RoboDK station: Config_1NewDrillbit.rdk

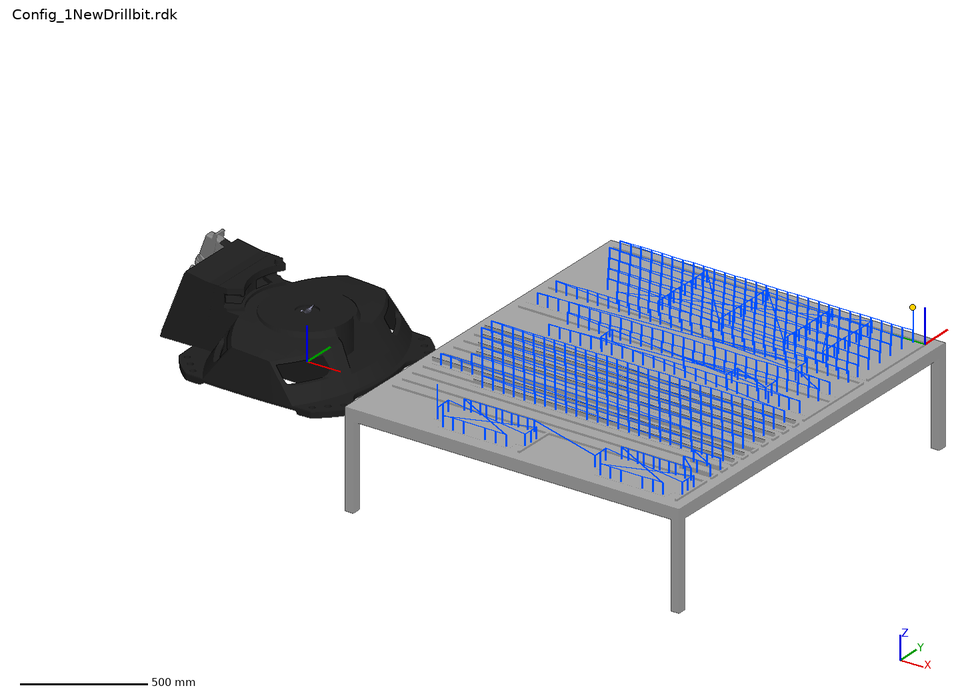
[picture v0: the station drawn from its stored meshes, robots at their saved joint values, targets as dots, program paths as lines]
Station Config_1NewDrillbit (saved by RoboDK 5.2.3). Poses are relative to the parent item; angles as X-Y-Z fixed-axis rotations.
  - frame KUKA KR 210 R2700 extra Base at (0, 0, 0) mm
    - robot KUKA KR 210 R2700 extra: 6 axes, payload 210 kg, reach 2696 mm, repeatability 0.06 mm, weight 1068 kg
        joint limits [-185, -140, -120, -350, -125, -350] to [185, -5, 155, 350, 125, 350]; home [0, -90, 90, 0, 0, 0]; saved at [43.451, -82.307, 119.902, -52.09, 33.269, 83.395]
      - tool Spindle, TCP at (32, 0, 260) mm, rotated rx 0 ry 39 rz 0 deg, size 157.3 x 72 x 259.9 mm
  - frame Corner First Plate at (2495, 660, 510.8) mm, rotated rx 0 ry 0 rz 90 deg
  - object Table 1 at (1700, -800, 455) mm, rotated rx 0 ry 0 rz 90 deg, size 1820 x 1600 x 475 mm, geometry from Table 1.stl
  - machining project Path1 settings: rotZ(0) | rotX(0)*rotY(0) | rotz(0) | onStart | onPathStart | onApproach | onPoint | onRetract | onFinish | SetRPM(%1) | SetTool(%1) | Extruder(%1) | default | default | OutOnMov(%1) | OutOffMov(%1) | onPathFinish | M_RunCode(%1)
  - program Path1 (1722 instructions, listed below)
  - object Config_1 at (2495, 660, 510.8) mm, rotated rx 0 ry 0 rz 90 deg
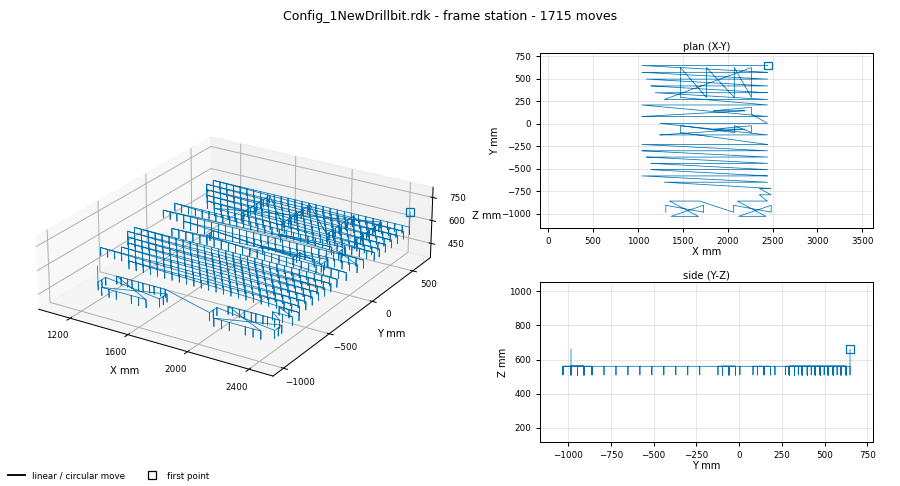
[picture p0: tool path of Config_1NewDrillbit.rdk in frame station, 1715 of 1715 moves have a stored position in this frame; points joined in program order, loops and branches not executed]

--- program Path1 (robot KUKA KR 210 R2700 extra) ---
  Smooth(1)
  Set speed (1000.0 mm/s)
  Set Ref.: Corner First Plate
  Set Tool: Spindle
  Show Spindle
  MoveJ 1 to (-10.8, 50, 150) mm, rotated rx -180 ry 0 rz 90 deg; joints [-16.649, -45.763, 65.757, 18.983, 33.662, -29.06]
  MoveL 2 to (-10.8, 50, 150) mm, rotated rx -180 ry 0 rz 90 deg; joints [-16.649, -45.763, 65.757, 18.983, 33.662, -29.06]
  MoveL 3 to (-10.8, 50, 50) mm, rotated rx -180 ry 0 rz 90 deg; joints [-16.649, -43.604, 67.207, 20.959, 30.27, -31.388]
  MoveL 4 to (-10.8, 50, 50) mm, rotated rx -180 ry 0 rz 90 deg; joints [-16.649, -43.604, 67.207, 20.959, 30.27, -31.388]
  Set speed (150.0 mm/s)
  MoveL 5 to (-10.8, 50, -0.5) mm, rotated rx 180 ry 0 rz 90 deg; joints [-16.649, -42.408, 67.766, 22.1, 28.636, -32.698]
  MoveL 6 to (-10.8, 50, 50) mm, rotated rx -180 ry 0 rz 90 deg; joints [-16.649, -43.604, 67.207, 20.959, 30.27, -31.388]
  MoveL 7 to (-10.8, 100, 50) mm, rotated rx 180 ry 0 rz 90 deg; joints [-17.019, -45.861, 71.178, 22.478, 28.801, -33.31]
  MoveL 8 to (-10.8, 100, -0.5) mm, rotated rx -180 ry 0 rz 90 deg; joints [-17.019, -44.622, 71.724, 23.798, 27.159, -34.805]
  MoveL 9 to (-10.8, 100, 50) mm, rotated rx 180 ry 0 rz 90 deg; joints [-17.019, -45.861, 71.178, 22.478, 28.801, -33.31]
  MoveL 10 to (-10.8, 150, 50) mm, rotated rx 180 ry 0 rz 90 deg; joints [-17.405, -48.034, 74.962, 24.095, 27.459, -35.336]
  MoveL 11 to (-10.8, 150, -0.5) mm, rotated rx 180 ry 0 rz 90 deg; joints [-17.405, -46.752, 75.499, 25.62, 25.808, -37.042]
  MoveL 12 to (-10.8, 150, 50) mm, rotated rx 180 ry 0 rz 90 deg; joints [-17.405, -48.034, 74.962, 24.095, 27.459, -35.336]
  MoveL 13 to (-10.8, 200, 50) mm, rotated rx -180 ry 0 rz 90 deg; joints [-17.809, -50.139, 78.585, 25.814, 26.233, -37.473]
  MoveL 14 to (-10.8, 200, -0.5) mm, rotated rx -180 ry 0 rz 90 deg; joints [-17.809, -48.813, 79.116, 27.569, 24.574, -39.416]
  MoveL 15 to (-10.8, 200, 50) mm, rotated rx -180 ry 0 rz 90 deg; joints [-17.809, -50.139, 78.585, 25.814, 26.233, -37.473]
  MoveL 16 to (-10.8, 250, 50) mm, rotated rx 180 ry 0 rz 90 deg; joints [-18.231, -52.185, 82.068, 27.636, 25.116, -39.724]
  MoveL 17 to (-10.8, 250, -0.5) mm, rotated rx 180 ry 0 rz 90 deg; joints [-18.231, -50.816, 82.594, 29.651, 23.452, -41.933]
  MoveL 18 to (-10.8, 250, 50) mm, rotated rx 180 ry 0 rz 90 deg; joints [-18.231, -52.185, 82.068, 27.636, 25.116, -39.724]
  MoveL 19 to (-10.8, 300, 50) mm, rotated rx -180 ry 0 rz 90 deg; joints [-18.673, -54.184, 85.426, 29.563, 24.104, -42.09]
  MoveL 20 to (-10.8, 300, -0.5) mm, rotated rx -180 ry 0 rz 90 deg; joints [-18.673, -52.769, 85.95, 31.865, 22.437, -44.595]
  MoveL 21 to (-10.8, 300, 50) mm, rotated rx -180 ry 0 rz 90 deg; joints [-18.673, -54.184, 85.426, 29.563, 24.104, -42.09]
  MoveL 22 to (-10.8, 350, 50) mm, rotated rx 180 ry 0 rz 90 deg; joints [-19.136, -56.141, 88.674, 31.59, 23.193, -44.569]
  MoveL 23 to (-10.8, 350, -0.5) mm, rotated rx 180 ry 0 rz 90 deg; joints [-19.136, -54.681, 89.197, 34.21, 21.527, -47.403]
  MoveL 24 to (-10.8, 350, 50) mm, rotated rx 180 ry 0 rz 90 deg; joints [-19.136, -56.141, 88.674, 31.59, 23.193, -44.569]
  MoveL 25 to (-10.8, 400, 50) mm, rotated rx -180 ry 0 rz 90 deg; joints [-19.622, -58.066, 91.821, 33.711, 22.382, -47.158]
  MoveL 26 to (-10.8, 400, -0.5) mm, rotated rx 180 ry 0 rz 90 deg; joints [-19.622, -56.557, 92.346, 36.679, 20.72, -50.348]
  MoveL 27 to (-10.8, 400, 50) mm, rotated rx -180 ry 0 rz 90 deg; joints [-19.622, -58.066, 91.821, 33.711, 22.382, -47.158]
  MoveL 28 to (-10.8, 450, 50) mm, rotated rx 180 ry 0 rz 90 deg; joints [-20.132, -59.962, 94.878, 35.915, 21.67, -49.846]
  MoveL 29 to (-10.8, 450, -0.5) mm, rotated rx -180 ry 0 rz 90 deg; joints [-20.132, -58.404, 95.405, 39.258, 20.016, -53.422]
  MoveL 30 to (-10.8, 450, 50) mm, rotated rx 180 ry 0 rz 90 deg; joints [-20.132, -59.962, 94.878, 35.915, 21.67, -49.846]
  MoveL 31 to (-10.8, 500, 50) mm, rotated rx 180 ry 0 rz 90 deg; joints [-20.668, -61.836, 97.851, 38.189, 21.056, -52.621]
  MoveL 32 to (-10.8, 500, -0.5) mm, rotated rx -180 ry 0 rz 90 deg; joints [-20.668, -60.227, 98.383, 41.928, 19.416, -56.606]
  MoveL 33 to (-10.8, 500, 50) mm, rotated rx 180 ry 0 rz 90 deg; joints [-20.668, -61.836, 97.851, 38.189, 21.056, -52.621]
  MoveL 34 to (-10.8, 550, 50) mm, rotated rx -180 ry 0 rz 90 deg; joints [-21.232, -63.693, 100.748, 40.512, 20.539, -55.465]
  MoveL 35 to (-10.8, 550, -0.5) mm, rotated rx 180 ry 0 rz 90 deg; joints [-21.232, -62.029, 101.285, 44.666, 18.917, -59.878]
  MoveL 36 to (-10.8, 550, 50) mm, rotated rx -180 ry 0 rz 90 deg; joints [-21.232, -63.693, 100.748, 40.512, 20.539, -55.465]
  MoveL 37 to (-10.8, 600, 50) mm, rotated rx 180 ry 0 rz 90 deg; joints [-21.826, -65.537, 103.573, 42.861, 20.119, -58.356]
  MoveL 38 to (-10.8, 600, -0.5) mm, rotated rx 180 ry 0 rz 90 deg; joints [-21.826, -63.817, 104.117, 47.441, 18.521, -63.209]
  MoveL 39 to (-10.8, 600, 50) mm, rotated rx 180 ry 0 rz 90 deg; joints [-21.826, -65.537, 103.573, 42.861, 20.119, -58.356]
  MoveL 40 to (-10.8, 650, 50) mm, rotated rx -180 ry 0 rz 90 deg; joints [-22.453, -67.372, 106.331, 45.208, 19.797, -61.269]
  MoveL 41 to (-10.8, 650, -0.5) mm, rotated rx 180 ry 0 rz 90 deg; joints [-22.453, -65.593, 106.883, 50.215, 18.227, -66.564]
  MoveL 42 to (-10.8, 650, 50) mm, rotated rx -180 ry 0 rz 90 deg; joints [-22.453, -67.372, 106.331, 45.208, 19.797, -61.269]
  MoveL 43 to (-10.8, 700, 50) mm, rotated rx -180 ry 0 rz 90 deg; joints [-23.115, -69.203, 109.025, 47.523, 19.571, -64.173]
  MoveL 44 to (-10.8, 700, -0.5) mm, rotated rx 180 ry 0 rz 90 deg; joints [-23.115, -67.362, 109.587, 52.95, 18.032, -69.905]
  MoveL 45 to (-10.8, 700, 50) mm, rotated rx -180 ry 0 rz 90 deg; joints [-23.115, -69.203, 109.025, 47.523, 19.571, -64.173]
  MoveL 46 to (-10.8, 750, 50) mm, rotated rx -180 ry 0 rz 90 deg; joints [-23.814, -71.033, 111.66, 49.773, 19.44, -67.039]
  MoveL 47 to (-10.8, 750, -0.5) mm, rotated rx 180 ry 0 rz 90 deg; joints [-23.814, -69.127, 112.233, 55.604, 17.936, -73.194]
  MoveL 48 to (-10.8, 750, 50) mm, rotated rx -180 ry 0 rz 90 deg; joints [-23.814, -71.033, 111.66, 49.773, 19.44, -67.039]
  MoveL 49 to (-10.8, 800, 50) mm, rotated rx -180 ry 0 rz 90 deg; joints [-24.555, -72.867, 114.238, 51.923, 19.404, -69.834]
  MoveL 50 to (-10.8, 800, -0.5) mm, rotated rx -180 ry 0 rz 90 deg; joints [-24.555, -70.893, 114.823, 58.134, 17.935, -76.388]
  MoveL 51 to (-10.8, 800, 50) mm, rotated rx -180 ry 0 rz 90 deg; joints [-24.555, -72.867, 114.238, 51.923, 19.404, -69.834]
  MoveL 52 to (-10.8, 850, 50) mm, rotated rx 180 ry 0 rz 90 deg; joints [-25.34, -74.708, 116.76, 53.942, 19.461, -72.529]
  MoveL 53 to (-10.8, 850, -0.5) mm, rotated rx 180 ry 0 rz 90 deg; joints [-25.34, -72.662, 117.358, 60.5, 18.027, -79.453]
  MoveL 54 to (-10.8, 850, 50) mm, rotated rx 180 ry 0 rz 90 deg; joints [-25.34, -74.708, 116.76, 53.942, 19.461, -72.529]
  MoveL 55 to (-10.8, 900, 50) mm, rotated rx -180 ry 0 rz 90 deg; joints [-26.173, -76.561, 119.228, 55.798, 19.61, -75.093]
  MoveL 56 to (-10.8, 900, -0.5) mm, rotated rx -180 ry 0 rz 90 deg; joints [-26.173, -74.439, 119.842, 62.666, 18.208, -82.352]
  MoveL 57 to (-10.8, 900, 50) mm, rotated rx -180 ry 0 rz 90 deg; joints [-26.173, -76.561, 119.228, 55.798, 19.61, -75.093]
  MoveL 58 to (-10.8, 950, 50) mm, rotated rx -180 ry 0 rz 90 deg; joints [-27.058, -78.43, 121.643, 57.462, 19.851, -77.502]
  MoveL 59 to (-10.8, 950, -0.5) mm, rotated rx 180 ry 0 rz 90 deg; joints [-27.058, -76.227, 122.274, 64.602, 18.476, -85.059]
  MoveL 60 to (-10.8, 950, 50) mm, rotated rx -180 ry 0 rz 90 deg; joints [-27.058, -78.43, 121.643, 57.462, 19.851, -77.502]
  MoveL 61 to (-10.8, 1000, 50) mm, rotated rx 180 ry 0 rz 90 deg; joints [-28.001, -80.318, 124.007, 58.912, 20.182, -79.735]
  MoveL 62 to (-10.8, 1000, -0.5) mm, rotated rx 180 ry 0 rz 90 deg; joints [-28.001, -78.031, 124.656, 66.28, 18.827, -87.549]
  MoveL 63 to (-10.8, 1000, 50) mm, rotated rx 180 ry 0 rz 90 deg; joints [-28.001, -80.318, 124.007, 58.912, 20.182, -79.735]
  MoveL 64 to (-10.8, 1050, 50) mm, rotated rx -180 ry 0 rz 90 deg; joints [-29.005, -82.231, 126.318, 60.129, 20.604, -81.776]
  MoveL 65 to (-10.8, 1050, -0.5) mm, rotated rx 180 ry 0 rz 90 deg; joints [-29.005, -79.854, 126.988, 67.681, 19.26, -89.808]
  MoveL 66 to (-10.8, 1050, 50) mm, rotated rx -180 ry 0 rz 90 deg; joints [-29.005, -82.231, 126.318, 60.129, 20.604, -81.776]
  MoveL 67 to (-10.8, 1100, 50) mm, rotated rx 180 ry 0 rz 90 deg; joints [-30.078, -84.172, 128.578, 61.097, 21.117, -83.613]
  MoveL 68 to (-10.8, 1100, -0.5) mm, rotated rx 180 ry 0 rz 90 deg; joints [-30.078, -81.701, 129.27, 68.792, 19.774, -91.823]
  MoveL 69 to (-10.8, 1100, 50) mm, rotated rx 180 ry 0 rz 90 deg; joints [-30.078, -84.172, 128.578, 61.097, 21.117, -83.613]
  MoveL 70 to (-10.8, 1150, 50) mm, rotated rx -180 ry 0 rz 90 deg; joints [-31.224, -86.147, 130.785, 61.808, 21.724, -85.24]
  MoveL 71 to (-10.8, 1150, -0.5) mm, rotated rx 180 ry 0 rz 90 deg; joints [-31.224, -83.576, 131.502, 69.603, 20.368, -93.59]
  MoveL 72 to (-10.8, 1150, 50) mm, rotated rx -180 ry 0 rz 90 deg; joints [-31.224, -86.147, 130.785, 61.808, 21.724, -85.24]
  MoveL 73 to (-10.8, 1200, 50) mm, rotated rx 180 ry 0 rz 90 deg; joints [-32.452, -88.16, 132.937, 62.257, 22.43, -86.657]
  MoveL 74 to (-10.8, 1200, -0.5) mm, rotated rx 180 ry 0 rz 90 deg; joints [-32.452, -85.485, 133.681, 70.11, 21.045, -95.109]
  MoveL 75 to (-10.8, 1200, 50) mm, rotated rx 180 ry 0 rz 90 deg; joints [-32.452, -88.16, 132.937, 62.257, 22.43, -86.657]
  MoveL 76 to (-10.8, 1250, 50) mm, rotated rx 180 ry 0 rz 90 deg; joints [-33.768, -90.216, 135.034, 62.444, 23.238, -87.866]
  MoveL 77 to (-10.8, 1250, -0.5) mm, rotated rx 180 ry 0 rz 90 deg; joints [-33.768, -87.431, 135.807, 70.315, 21.808, -96.384]
  MoveL 78 to (-10.8, 1250, 50) mm, rotated rx 180 ry 0 rz 90 deg; joints [-33.768, -90.216, 135.034, 62.444, 23.238, -87.866]
  MoveL 79 to (-10.8, 1300, 50) mm, rotated rx 180 ry 0 rz 90 deg; joints [-35.181, -92.32, 137.073, 62.376, 24.157, -88.879]
  MoveL 80 to (-10.8, 1300, -0.5) mm, rotated rx -180 ry 0 rz 90 deg; joints [-35.181, -89.419, 137.878, 70.222, 22.664, -97.425]
  MoveL 81 to (-10.8, 1300, 50) mm, rotated rx 180 ry 0 rz 90 deg; joints [-35.181, -92.32, 137.073, 62.376, 24.157, -88.879]
  MoveL 82 to (-10.8, 1350, 50) mm, rotated rx -180 ry 0 rz 90 deg; joints [-36.701, -94.476, 139.051, 62.061, 25.197, -89.708]
  MoveL 83 to (-10.8, 1350, -0.5) mm, rotated rx -180 ry 0 rz 90 deg; joints [-36.701, -91.455, 139.89, 69.839, 23.619, -98.245]
  MoveL 84 to (-10.8, 1350, 50) mm, rotated rx -180 ry 0 rz 90 deg; joints [-36.701, -94.476, 139.051, 62.061, 25.197, -89.708]
  MoveL 85 to (-10.8, 1400, 50) mm, rotated rx -180 ry 0 rz 90 deg; joints [-38.337, -96.689, 140.964, 61.514, 26.367, -90.372]
  MoveL 86 to (-10.8, 1400, -0.5) mm, rotated rx 180 ry 0 rz 90 deg; joints [-38.337, -93.543, 141.842, 69.179, 24.685, -98.863]
  MoveL 87 to (-10.8, 1400, 50) mm, rotated rx -180 ry 0 rz 90 deg; joints [-38.337, -96.689, 140.964, 61.514, 26.367, -90.372]
  MoveL 88 to (-10.8, 1450, 50) mm, rotated rx -180 ry 0 rz 90 deg; joints [-40.1, -98.961, 142.81, 60.755, 27.683, -90.897]
  MoveL 89 to (-10.8, 1450, -0.5) mm, rotated rx -180 ry 0 rz 90 deg; joints [-40.1, -95.687, 143.728, 68.26, 25.874, -99.3]
  MoveL 90 to (-10.8, 1450, 50) mm, rotated rx -180 ry 0 rz 90 deg; joints [-40.1, -98.961, 142.81, 60.755, 27.683, -90.897]
  MoveL 91 to (-86.48, 50, 50) mm, rotated rx 180 ry 0 rz 90 deg; joints [-14.798, -44.582, 68.933, 19.373, 28.984, -28.699]
  MoveL 92 to (-86.48, 50, -0.5) mm, rotated rx 180 ry 0 rz 90 deg; joints [-14.798, -43.367, 69.486, 20.5, 27.322, -29.977]
  MoveL 93 to (-86.48, 50, 50) mm, rotated rx 180 ry 0 rz 90 deg; joints [-14.798, -44.582, 68.933, 19.373, 28.984, -28.699]
  MoveL 94 to (-86.48, 100, 50) mm, rotated rx 180 ry 0 rz 90 deg; joints [-15.131, -46.823, 72.859, 20.836, 27.506, -30.521]
  MoveL 95 to (-86.48, 100, -0.5) mm, rotated rx -180 ry 0 rz 90 deg; joints [-15.131, -45.565, 73.401, 22.149, 25.831, -31.99]
  MoveL 96 to (-86.48, 100, 50) mm, rotated rx 180 ry 0 rz 90 deg; joints [-15.131, -46.823, 72.859, 20.836, 27.506, -30.521]
  MoveL 97 to (-86.48, 150, 50) mm, rotated rx -180 ry 0 rz 90 deg; joints [-15.479, -48.988, 76.608, 22.405, 26.146, -32.455]
  MoveL 98 to (-86.48, 150, -0.5) mm, rotated rx -180 ry 0 rz 90 deg; joints [-15.479, -47.686, 77.142, 23.933, 24.459, -34.144]
  MoveL 99 to (-86.48, 150, 50) mm, rotated rx -180 ry 0 rz 90 deg; joints [-15.479, -48.988, 76.608, 22.405, 26.146, -32.455]
  MoveL 100 to (-86.48, 200, 50) mm, rotated rx -180 ry 0 rz 90 deg; joints [-15.843, -51.088, 80.205, 24.086, 24.897, -34.509]
  MoveL 101 to (-86.48, 200, -0.5) mm, rotated rx 180 ry 0 rz 90 deg; joints [-15.843, -49.742, 80.734, 25.859, 23.198, -36.45]
  MoveL 102 to (-86.48, 200, 50) mm, rotated rx -180 ry 0 rz 90 deg; joints [-15.843, -51.088, 80.205, 24.086, 24.897, -34.509]
  MoveL 103 to (-86.48, 250, 50) mm, rotated rx 180 ry 0 rz 90 deg; joints [-16.224, -53.135, 83.669, 25.883, 23.753, -36.689]
  MoveL 104 to (-86.48, 250, -0.5) mm, rotated rx -180 ry 0 rz 90 deg; joints [-16.224, -51.744, 84.194, 27.935, 22.045, -38.917]
  MoveL 105 to (-86.48, 250, 50) mm, rotated rx 180 ry 0 rz 90 deg; joints [-16.224, -53.135, 83.669, 25.883, 23.753, -36.689]
  MoveL 106 to (-86.48, 300, 50) mm, rotated rx -180 ry 0 rz 90 deg; joints [-16.624, -55.137, 87.014, 27.798, 22.709, -38.998]
  MoveL 107 to (-86.48, 300, -0.5) mm, rotated rx 180 ry 0 rz 90 deg; joints [-16.624, -53.701, 87.537, 30.167, 20.994, -41.55]
  MoveL 108 to (-86.48, 300, 50) mm, rotated rx -180 ry 0 rz 90 deg; joints [-16.624, -55.137, 87.014, 27.798, 22.709, -38.998]
  MoveL 109 to (-86.48, 350, 50) mm, rotated rx 180 ry 0 rz 90 deg; joints [-17.042, -57.103, 90.253, 29.831, 21.764, -41.437]
  MoveL 110 to (-86.48, 350, -0.5) mm, rotated rx 180 ry 0 rz 90 deg; joints [-17.042, -55.619, 90.777, 32.555, 20.045, -44.353]
  MoveL 111 to (-86.48, 350, 50) mm, rotated rx 180 ry 0 rz 90 deg; joints [-17.042, -57.103, 90.253, 29.831, 21.764, -41.437]
  MoveL 112 to (-86.48, 400, 50) mm, rotated rx 180 ry 0 rz 90 deg; joints [-17.482, -59.039, 93.396, 31.978, 20.915, -44.004]
  MoveL 113 to (-86.48, 400, -0.5) mm, rotated rx 180 ry 0 rz 90 deg; joints [-17.482, -57.506, 93.922, 35.095, 19.197, -47.323]
  MoveL 114 to (-86.48, 400, 50) mm, rotated rx 180 ry 0 rz 90 deg; joints [-17.482, -59.039, 93.396, 31.978, 20.915, -44.004]
  MoveL 115 to (-86.48, 450, 50) mm, rotated rx -180 ry 0 rz 90 deg; joints [-17.945, -60.951, 96.453, 34.23, 20.163, -46.692]
  MoveL 116 to (-86.48, 450, -0.5) mm, rotated rx 180 ry 0 rz 90 deg; joints [-17.945, -59.366, 96.983, 37.779, 18.451, -50.452]
  MoveL 117 to (-86.48, 450, 50) mm, rotated rx -180 ry 0 rz 90 deg; joints [-17.945, -60.951, 96.453, 34.23, 20.163, -46.692]
  MoveL 118 to (-86.48, 500, 50) mm, rotated rx 180 ry 0 rz 90 deg; joints [-18.431, -62.844, 99.43, 36.574, 19.507, -49.488]
  MoveL 119 to (-86.48, 500, -0.5) mm, rotated rx 180 ry 0 rz 90 deg; joints [-18.431, -61.206, 99.965, 40.589, 17.807, -53.725]
  MoveL 120 to (-86.48, 500, 50) mm, rotated rx 180 ry 0 rz 90 deg; joints [-18.431, -62.844, 99.43, 36.574, 19.507, -49.488]
  MoveL 121 to (-86.48, 550, 50) mm, rotated rx 180 ry 0 rz 90 deg; joints [-18.944, -64.724, 102.334, 38.99, 18.948, -52.374]
  MoveL 122 to (-86.48, 550, -0.5) mm, rotated rx -180 ry 0 rz 90 deg; joints [-18.944, -63.029, 102.875, 43.499, 17.266, -57.118]
  MoveL 123 to (-86.48, 550, 50) mm, rotated rx 180 ry 0 rz 90 deg; joints [-18.944, -64.724, 102.334, 38.99, 18.948, -52.374]
  MoveL 124 to (-86.48, 600, 50) mm, rotated rx -180 ry 0 rz 90 deg; joints [-19.485, -66.595, 105.169, 41.455, 18.486, -55.329]
  MoveL 125 to (-86.48, 600, -0.5) mm, rotated rx -180 ry 0 rz 90 deg; joints [-19.485, -64.841, 105.718, 46.478, 16.828, -60.599]
  MoveL 126 to (-86.48, 600, 50) mm, rotated rx -180 ry 0 rz 90 deg; joints [-19.485, -66.595, 105.169, 41.455, 18.486, -55.329]
  MoveL 127 to (-86.48, 650, 50) mm, rotated rx 180 ry 0 rz 90 deg; joints [-20.056, -68.461, 107.941, 43.937, 18.122, -58.322]
  MoveL 128 to (-86.48, 650, -0.5) mm, rotated rx 180 ry 0 rz 90 deg; joints [-20.056, -66.646, 108.498, 49.483, 16.493, -64.13]
  MoveL 129 to (-86.48, 650, 50) mm, rotated rx 180 ry 0 rz 90 deg; joints [-20.056, -68.461, 107.941, 43.937, 18.122, -58.322]
  MoveL 130 to (-86.48, 700, 50) mm, rotated rx -180 ry 0 rz 90 deg; joints [-20.661, -70.327, 110.652, 46.401, 17.855, -61.321]
  MoveL 131 to (-86.48, 700, -0.5) mm, rotated rx 180 ry 0 rz 90 deg; joints [-20.661, -68.447, 111.22, 52.467, 16.26, -67.665]
  MoveL 132 to (-86.48, 700, 50) mm, rotated rx -180 ry 0 rz 90 deg; joints [-20.661, -70.327, 110.652, 46.401, 17.855, -61.321]
  MoveL 133 to (-86.48, 750, 50) mm, rotated rx -180 ry 0 rz 90 deg; joints [-21.301, -72.199, 113.306, 48.809, 17.686, -64.288]
  MoveL 134 to (-86.48, 750, -0.5) mm, rotated rx 180 ry 0 rz 90 deg; joints [-21.301, -70.25, 113.886, 55.379, 16.129, -71.153]
  MoveL 135 to (-86.48, 750, 50) mm, rotated rx -180 ry 0 rz 90 deg; joints [-21.301, -72.199, 113.306, 48.809, 17.686, -64.288]
  MoveL 136 to (-86.48, 800, 50) mm, rotated rx -180 ry 0 rz 90 deg; joints [-21.98, -74.079, 115.905, 51.119, 17.613, -67.184]
  MoveL 137 to (-86.48, 800, -0.5) mm, rotated rx -180 ry 0 rz 90 deg; joints [-21.98, -72.058, 116.499, 58.165, 16.096, -74.544]
  MoveL 138 to (-86.48, 800, 50) mm, rotated rx -180 ry 0 rz 90 deg; joints [-21.98, -74.079, 115.905, 51.119, 17.613, -67.184]
  MoveL 139 to (-86.48, 850, 50) mm, rotated rx 180 ry 0 rz 90 deg; joints [-22.702, -75.973, 118.452, 53.291, 17.635, -69.971]
  MoveL 140 to (-86.48, 850, -0.5) mm, rotated rx -180 ry 0 rz 90 deg; joints [-22.702, -73.875, 119.061, 60.773, 16.159, -77.789]
  MoveL 141 to (-86.48, 850, 50) mm, rotated rx 180 ry 0 rz 90 deg; joints [-22.702, -75.973, 118.452, 53.291, 17.635, -69.971]
  MoveL 142 to (-86.48, 900, 50) mm, rotated rx 180 ry 0 rz 90 deg; joints [-23.469, -77.886, 120.948, 55.285, 17.752, -72.611]
  MoveL 143 to (-86.48, 900, -0.5) mm, rotated rx 180 ry 0 rz 90 deg; joints [-23.469, -75.707, 121.574, 63.158, 16.314, -80.843]
  MoveL 144 to (-86.48, 900, 50) mm, rotated rx 180 ry 0 rz 90 deg; joints [-23.469, -77.886, 120.948, 55.285, 17.752, -72.611]
  MoveL 145 to (-86.48, 950, 50) mm, rotated rx -180 ry 0 rz 90 deg; joints [-24.288, -79.823, 123.395, 57.066, 17.964, -75.072]
  MoveL 146 to (-86.48, 950, -0.5) mm, rotated rx -180 ry 0 rz 90 deg; joints [-24.288, -77.558, 124.039, 65.278, 16.557, -83.669]
  MoveL 147 to (-86.48, 950, 50) mm, rotated rx -180 ry 0 rz 90 deg; joints [-24.288, -79.823, 123.395, 57.066, 17.964, -75.072]
  MoveL 148 to (-86.48, 1000, 50) mm, rotated rx -180 ry 0 rz 90 deg; joints [-25.161, -81.788, 125.791, 58.604, 18.268, -77.326]
  MoveL 149 to (-86.48, 1000, -0.5) mm, rotated rx 180 ry 0 rz 90 deg; joints [-25.161, -79.433, 126.457, 67.099, 16.885, -86.235]
  MoveL 150 to (-86.48, 1000, 50) mm, rotated rx -180 ry 0 rz 90 deg; joints [-25.161, -81.788, 125.791, 58.604, 18.268, -77.326]
  MoveL 151 to (-86.48, 1050, 50) mm, rotated rx -180 ry 0 rz 90 deg; joints [-26.095, -83.789, 128.139, 59.872, 18.666, -79.349]
  MoveL 152 to (-86.48, 1050, -0.5) mm, rotated rx -180 ry 0 rz 90 deg; joints [-26.095, -81.337, 128.827, 68.595, 17.297, -88.518]
  MoveL 153 to (-86.48, 1050, 50) mm, rotated rx -180 ry 0 rz 90 deg; joints [-26.095, -83.789, 128.139, 59.872, 18.666, -79.349]
  MoveL 154 to (-86.48, 1100, 50) mm, rotated rx 180 ry 0 rz 90 deg; joints [-27.096, -85.831, 130.438, 60.853, 19.16, -81.127]
  MoveL 155 to (-86.48, 1100, -0.5) mm, rotated rx -180 ry 0 rz 90 deg; joints [-27.096, -83.277, 131.151, 69.748, 17.79, -90.503]
  MoveL 156 to (-86.48, 1100, 50) mm, rotated rx 180 ry 0 rz 90 deg; joints [-27.096, -85.831, 130.438, 60.853, 19.16, -81.127]
  MoveL 157 to (-86.48, 1150, 50) mm, rotated rx -180 ry 0 rz 90 deg; joints [-28.17, -87.921, 132.686, 61.533, 19.753, -82.65]
  MoveL 158 to (-86.48, 1150, -0.5) mm, rotated rx -180 ry 0 rz 90 deg; joints [-28.17, -85.258, 133.427, 70.547, 18.366, -92.183]
  MoveL 159 to (-86.48, 1150, 50) mm, rotated rx -180 ry 0 rz 90 deg; joints [-28.17, -87.921, 132.686, 61.533, 19.753, -82.65]
  MoveL 160 to (-86.48, 1200, 50) mm, rotated rx 180 ry 0 rz 90 deg; joints [-29.325, -90.065, 134.884, 61.907, 20.45, -83.915]
  MoveL 161 to (-86.48, 1200, -0.5) mm, rotated rx 180 ry 0 rz 90 deg; joints [-29.325, -87.288, 135.655, 70.984, 19.027, -93.555]
  MoveL 162 to (-86.48, 1200, 50) mm, rotated rx 180 ry 0 rz 90 deg; joints [-29.325, -90.065, 134.884, 61.907, 20.45, -83.915]
  MoveL 163 to (-86.48, 1250, 50) mm, rotated rx 180 ry 0 rz 90 deg; joints [-30.57, -92.272, 137.028, 61.975, 21.259, -84.926]
  MoveL 164 to (-86.48, 1250, -0.5) mm, rotated rx 180 ry 0 rz 90 deg; joints [-30.57, -89.374, 137.832, 71.061, 19.778, -94.623]
  MoveL 165 to (-86.48, 1250, 50) mm, rotated rx 180 ry 0 rz 90 deg; joints [-30.57, -92.272, 137.028, 61.975, 21.259, -84.926]
  MoveL 166 to (-86.48, 1300, 50) mm, rotated rx 180 ry 0 rz 90 deg; joints [-31.913, -94.55, 139.117, 61.744, 22.19, -85.693]
  MoveL 167 to (-86.48, 1300, -0.5) mm, rotated rx -180 ry 0 rz 90 deg; joints [-31.913, -91.525, 139.957, 70.782, 20.629, -95.397]
  MoveL 168 to (-86.48, 1300, 50) mm, rotated rx 180 ry 0 rz 90 deg; joints [-31.913, -94.55, 139.117, 61.744, 22.19, -85.693]
  MoveL 169 to (-86.48, 1350, 50) mm, rotated rx 180 ry 0 rz 90 deg; joints [-33.365, -96.907, 141.147, 61.226, 23.258, -86.233]
  MoveL 170 to (-86.48, 1350, -0.5) mm, rotated rx -180 ry 0 rz 90 deg; joints [-33.365, -93.749, 142.028, 70.158, 21.589, -95.891]
  MoveL 171 to (-86.48, 1350, 50) mm, rotated rx 180 ry 0 rz 90 deg; joints [-33.365, -96.907, 141.147, 61.226, 23.258, -86.233]
  MoveL 172 to (-86.48, 1400, 50) mm, rotated rx -180 ry 0 rz 90 deg; joints [-34.939, -99.35, 143.114, 60.44, 24.478, -86.569]
  MoveL 173 to (-86.48, 1400, -0.5) mm, rotated rx -180 ry 0 rz 90 deg; joints [-34.939, -96.055, 144.039, 69.205, 22.676, -96.127]
  MoveL 174 to (-86.48, 1400, 50) mm, rotated rx -180 ry 0 rz 90 deg; joints [-34.939, -99.35, 143.114, 60.44, 24.478, -86.569]
  MoveL 175 to (-86.48, 1450, 50) mm, rotated rx 180 ry 0 rz 90 deg; joints [-36.646, -101.889, 145.015, 59.412, 25.871, -86.731]
  MoveL 176 to (-86.48, 1450, -0.5) mm, rotated rx -180 ry 0 rz 90 deg; joints [-36.646, -98.452, 145.988, 67.945, 23.909, -96.132]
  MoveL 177 to (-86.48, 1450, 50) mm, rotated rx 180 ry 0 rz 90 deg; joints [-36.646, -101.889, 145.015, 59.412, 25.871, -86.731]
  MoveL 178 to (-162.16, 50, 50) mm, rotated rx 180 ry 0 rz 90 deg; joints [-12.916, -45.433, 70.428, 17.535, 27.831, -25.717]
  MoveL 179 to (-162.16, 50, -0.5) mm, rotated rx 180 ry 0 rz 90 deg; joints [-12.916, -44.202, 70.977, 18.62, 26.139, -26.934]
  MoveL 180 to (-162.16, 50, 50) mm, rotated rx 180 ry 0 rz 90 deg; joints [-12.916, -45.433, 70.428, 17.535, 27.831, -25.717]
  MoveL 181 to (-162.16, 100, 50) mm, rotated rx 180 ry 0 rz 90 deg; joints [-13.21, -47.663, 74.318, 18.914, 26.337, -27.409]
  MoveL 182 to (-162.16, 100, -0.5) mm, rotated rx 180 ry 0 rz 90 deg; joints [-13.21, -46.388, 74.857, 20.187, 24.628, -28.819]
  MoveL 183 to (-162.16, 100, 50) mm, rotated rx 180 ry 0 rz 90 deg; joints [-13.21, -47.663, 74.318, 18.914, 26.337, -27.409]
  MoveL 184 to (-162.16, 150, 50) mm, rotated rx 180 ry 0 rz 90 deg; joints [-13.517, -49.821, 78.04, 20.404, 24.955, -29.218]
  MoveL 185 to (-162.16, 150, -0.5) mm, rotated rx 180 ry 0 rz 90 deg; joints [-13.517, -48.502, 78.572, 21.897, 23.23, -30.854]
  MoveL 186 to (-162.16, 150, 50) mm, rotated rx 180 ry 0 rz 90 deg; joints [-13.517, -49.821, 78.04, 20.404, 24.955, -29.218]
  MoveL 187 to (-162.16, 200, 50) mm, rotated rx 180 ry 0 rz 90 deg; joints [-13.839, -51.919, 81.617, 22.012, 23.679, -31.154]
  MoveL 188 to (-162.16, 200, -0.5) mm, rotated rx 180 ry 0 rz 90 deg; joints [-13.839, -50.556, 82.144, 23.761, 21.937, -33.051]
  MoveL 189 to (-162.16, 200, 50) mm, rotated rx 180 ry 0 rz 90 deg; joints [-13.839, -51.919, 81.617, 22.012, 23.679, -31.154]
  MoveL 190 to (-162.16, 250, 50) mm, rotated rx 180 ry 0 rz 90 deg; joints [-14.176, -53.968, 85.066, 23.747, 22.502, -33.225]
  MoveL 191 to (-162.16, 250, -0.5) mm, rotated rx 180 ry 0 rz 90 deg; joints [-14.176, -52.558, 85.59, 25.791, 20.746, -35.423]
  MoveL 192 to (-162.16, 250, 50) mm, rotated rx 180 ry 0 rz 90 deg; joints [-14.176, -53.968, 85.066, 23.747, 22.502, -33.225]
  MoveL 193 to (-162.16, 300, 50) mm, rotated rx -180 ry 0 rz 90 deg; joints [-14.529, -55.976, 88.401, 25.613, 21.422, -35.437]
  MoveL 194 to (-162.16, 300, -0.5) mm, rotated rx 180 ry 0 rz 90 deg; joints [-14.529, -54.519, 88.924, 27.996, 19.654, -37.983]
  MoveL 195 to (-162.16, 300, 50) mm, rotated rx -180 ry 0 rz 90 deg; joints [-14.529, -55.976, 88.401, 25.613, 21.422, -35.437]
  MoveL 196 to (-162.16, 350, 50) mm, rotated rx 180 ry 0 rz 90 deg; joints [-14.901, -57.951, 91.634, 27.612, 20.435, -37.795]
  MoveL 197 to (-162.16, 350, -0.5) mm, rotated rx -180 ry 0 rz 90 deg; joints [-14.901, -56.445, 92.159, 30.385, 18.659, -40.737]
  MoveL 198 to (-162.16, 350, 50) mm, rotated rx 180 ry 0 rz 90 deg; joints [-14.901, -57.951, 91.634, 27.612, 20.435, -37.795]
  MoveL 199 to (-162.16, 400, 50) mm, rotated rx 180 ry 0 rz 90 deg; joints [-15.291, -59.898, 94.776, 29.745, 19.542, -40.299]
  MoveL 200 to (-162.16, 400, -0.5) mm, rotated rx 180 ry 0 rz 90 deg; joints [-15.291, -58.342, 95.304, 32.958, 17.762, -43.689]
  MoveL 201 to (-162.16, 400, 50) mm, rotated rx 180 ry 0 rz 90 deg; joints [-15.291, -59.898, 94.776, 29.745, 19.542, -40.299]
  MoveL 202 to (-162.16, 450, 50) mm, rotated rx -180 ry 0 rz 90 deg; joints [-15.702, -61.826, 97.835, 32.007, 18.743, -42.945]
  MoveL 203 to (-162.16, 450, -0.5) mm, rotated rx -180 ry 0 rz 90 deg; joints [-15.702, -60.216, 98.366, 35.712, 16.964, -46.837]
  MoveL 204 to (-162.16, 450, 50) mm, rotated rx -180 ry 0 rz 90 deg; joints [-15.702, -61.826, 97.835, 32.007, 18.743, -42.945]
  MoveL 205 to (-162.16, 500, 50) mm, rotated rx 180 ry 0 rz 90 deg; joints [-16.134, -63.737, 100.817, 34.388, 18.038, -45.725]
  MoveL 206 to (-162.16, 500, -0.5) mm, rotated rx 180 ry 0 rz 90 deg; joints [-16.134, -62.073, 101.354, 38.635, 16.266, -50.169]
  MoveL 207 to (-162.16, 500, 50) mm, rotated rx 180 ry 0 rz 90 deg; joints [-16.134, -63.737, 100.817, 34.388, 18.038, -45.725]
  MoveL 208 to (-162.16, 550, 50) mm, rotated rx 180 ry 0 rz 90 deg; joints [-16.591, -65.639, 103.728, 36.869, 17.427, -48.622]
  MoveL 209 to (-162.16, 550, -0.5) mm, rotated rx 180 ry 0 rz 90 deg; joints [-16.591, -63.916, 104.273, 41.703, 15.671, -53.664]
  MoveL 210 to (-162.16, 550, 50) mm, rotated rx 180 ry 0 rz 90 deg; joints [-16.591, -65.639, 103.728, 36.869, 17.427, -48.622]
  MoveL 211 to (-162.16, 600, 50) mm, rotated rx 180 ry 0 rz 90 deg; joints [-17.073, -67.536, 106.574, 39.426, 16.914, -51.614]
  MoveL 212 to (-162.16, 600, -0.5) mm, rotated rx -180 ry 0 rz 90 deg; joints [-17.073, -65.752, 107.127, 44.883, 15.179, -57.29]
  MoveL 213 to (-162.16, 600, 50) mm, rotated rx 180 ry 0 rz 90 deg; joints [-17.073, -67.536, 106.574, 39.426, 16.914, -51.614]
  MoveL 214 to (-162.16, 650, 50) mm, rotated rx 180 ry 0 rz 90 deg; joints [-17.584, -69.432, 109.359, 42.029, 16.497, -54.669]
  MoveL 215 to (-162.16, 650, -0.5) mm, rotated rx 180 ry 0 rz 90 deg; joints [-17.584, -67.583, 109.922, 48.13, 14.792, -61.005]
  MoveL 216 to (-162.16, 650, 50) mm, rotated rx 180 ry 0 rz 90 deg; joints [-17.584, -69.432, 109.359, 42.029, 16.497, -54.669]
  MoveL 217 to (-162.16, 700, 50) mm, rotated rx 180 ry 0 rz 90 deg; joints [-18.124, -71.333, 112.086, 44.636, 16.179, -57.751]
  MoveL 218 to (-162.16, 700, -0.5) mm, rotated rx -180 ry 0 rz 90 deg; joints [-18.124, -69.416, 112.661, 51.39, 14.509, -64.753]
  MoveL 219 to (-162.16, 700, 50) mm, rotated rx 180 ry 0 rz 90 deg; joints [-18.124, -71.333, 112.086, 44.636, 16.179, -57.751]
  MoveL 220 to (-162.16, 750, 50) mm, rotated rx 180 ry 0 rz 90 deg; joints [-18.698, -73.244, 114.759, 47.204, 15.959, -60.817]
  MoveL 221 to (-162.16, 750, -0.5) mm, rotated rx -180 ry 0 rz 90 deg; joints [-18.698, -71.255, 115.347, 54.597, 14.331, -68.474]
  MoveL 222 to (-162.16, 750, 50) mm, rotated rx 180 ry 0 rz 90 deg; joints [-18.698, -73.244, 114.759, 47.204, 15.959, -60.817]
  MoveL 223 to (-162.16, 800, 50) mm, rotated rx 180 ry 0 rz 90 deg; joints [-19.308, -75.169, 117.38, 49.683, 15.837, -63.817]
  MoveL 224 to (-162.16, 800, -0.5) mm, rotated rx -180 ry 0 rz 90 deg; joints [-19.308, -73.104, 117.982, 57.686, 14.254, -72.103]
  MoveL 225 to (-162.16, 800, 50) mm, rotated rx 180 ry 0 rz 90 deg; joints [-19.308, -75.169, 117.38, 49.683, 15.837, -63.817]
  MoveL 226 to (-162.16, 850, 50) mm, rotated rx -180 ry 0 rz 90 deg; joints [-19.958, -77.114, 119.951, 52.022, 15.814, -66.704]
  MoveL 227 to (-162.16, 850, -0.5) mm, rotated rx -180 ry 0 rz 90 deg; joints [-19.958, -74.969, 120.57, 60.589, 14.276, -75.573]
  MoveL 228 to (-162.16, 850, 50) mm, rotated rx -180 ry 0 rz 90 deg; joints [-19.958, -77.114, 119.951, 52.022, 15.814, -66.704]
  MoveL 229 to (-162.16, 900, 50) mm, rotated rx -180 ry 0 rz 90 deg; joints [-20.651, -79.086, 122.474, 54.171, 15.887, -69.43]
  MoveL 230 to (-162.16, 900, -0.5) mm, rotated rx 180 ry 0 rz 90 deg; joints [-20.651, -76.854, 123.111, 63.242, 14.392, -78.826]
  MoveL 231 to (-162.16, 900, 50) mm, rotated rx -180 ry 0 rz 90 deg; joints [-20.651, -79.086, 122.474, 54.171, 15.887, -69.43]
  MoveL 232 to (-162.16, 950, 50) mm, rotated rx -180 ry 0 rz 90 deg; joints [-21.391, -81.089, 124.949, 56.083, 16.057, -71.951]
  MoveL 233 to (-162.16, 950, -0.5) mm, rotated rx 180 ry 0 rz 90 deg; joints [-21.391, -78.766, 125.607, 65.592, 14.599, -81.807]
  MoveL 234 to (-162.16, 950, 50) mm, rotated rx -180 ry 0 rz 90 deg; joints [-21.391, -81.089, 124.949, 56.083, 16.057, -71.951]
  MoveL 235 to (-162.16, 1000, 50) mm, rotated rx -180 ry 0 rz 90 deg; joints [-22.183, -83.131, 127.378, 57.719, 16.323, -74.228]
  MoveL 236 to (-162.16, 1000, -0.5) mm, rotated rx -180 ry 0 rz 90 deg; joints [-22.183, -80.711, 128.058, 67.591, 14.893, -84.475]
  MoveL 237 to (-162.16, 1000, 50) mm, rotated rx -180 ry 0 rz 90 deg; joints [-22.183, -83.131, 127.378, 57.719, 16.323, -74.228]
  MoveL 238 to (-162.16, 1050, 50) mm, rotated rx -180 ry 0 rz 90 deg; joints [-23.033, -85.22, 129.76, 59.044, 16.686, -76.23]
  MoveL 239 to (-162.16, 1050, -0.5) mm, rotated rx -180 ry 0 rz 90 deg; joints [-23.033, -82.697, 130.466, 69.205, 15.271, -86.797]
  MoveL 240 to (-162.16, 1050, 50) mm, rotated rx -180 ry 0 rz 90 deg; joints [-23.033, -85.22, 129.76, 59.044, 16.686, -76.23]
  MoveL 241 to (-162.16, 1100, 50) mm, rotated rx -180 ry 0 rz 90 deg; joints [-23.947, -87.363, 132.096, 60.033, 17.149, -77.935]
  MoveL 242 to (-162.16, 1100, -0.5) mm, rotated rx -180 ry 0 rz 90 deg; joints [-23.947, -84.729, 132.829, 70.409, 15.732, -88.75]
  MoveL 243 to (-162.16, 1100, 50) mm, rotated rx -180 ry 0 rz 90 deg; joints [-23.947, -87.363, 132.096, 60.033, 17.149, -77.935]
  MoveL 244 to (-162.16, 1150, 50) mm, rotated rx -180 ry 0 rz 90 deg; joints [-24.932, -89.569, 134.385, 60.67, 17.716, -79.329]
  MoveL 245 to (-162.16, 1150, -0.5) mm, rotated rx 180 ry 0 rz 90 deg; joints [-24.932, -86.819, 135.149, 71.185, 16.276, -90.321]
  MoveL 246 to (-162.16, 1150, 50) mm, rotated rx -180 ry 0 rz 90 deg; joints [-24.932, -89.569, 134.385, 60.67, 17.716, -79.329]
  MoveL 247 to (-162.16, 1200, 50) mm, rotated rx 180 ry 0 rz 90 deg; joints [-25.995, -91.849, 136.625, 60.944, 18.393, -80.406]
  MoveL 248 to (-162.16, 1200, -0.5) mm, rotated rx -180 ry 0 rz 90 deg; joints [-25.995, -88.974, 137.423, 71.525, 16.907, -91.505]
  MoveL 249 to (-162.16, 1200, 50) mm, rotated rx 180 ry 0 rz 90 deg; joints [-25.995, -91.849, 136.625, 60.944, 18.393, -80.406]
  MoveL 250 to (-162.16, 1250, 50) mm, rotated rx 180 ry 0 rz 90 deg; joints [-27.146, -94.212, 138.815, 60.856, 19.193, -81.168]
  MoveL 251 to (-162.16, 1250, -0.5) mm, rotated rx -180 ry 0 rz 90 deg; joints [-27.146, -91.206, 139.65, 71.428, 17.632, -92.306]
  MoveL 252 to (-162.16, 1250, 50) mm, rotated rx 180 ry 0 rz 90 deg; joints [-27.146, -94.212, 138.815, 60.856, 19.193, -81.168]
  MoveL 253 to (-162.16, 1300, 50) mm, rotated rx -180 ry 0 rz 90 deg; joints [-28.395, -96.673, 140.951, 60.415, 20.129, -81.628]
  MoveL 254 to (-162.16, 1300, -0.5) mm, rotated rx 180 ry 0 rz 90 deg; joints [-28.395, -93.529, 141.828, 70.899, 18.464, -92.73]
  MoveL 255 to (-162.16, 1300, 50) mm, rotated rx -180 ry 0 rz 90 deg; joints [-28.395, -96.673, 140.951, 60.415, 20.129, -81.628]
  MoveL 256 to (-162.16, 1350, 50) mm, rotated rx 180 ry 0 rz 90 deg; joints [-29.753, -99.244, 143.032, 59.637, 21.22, -81.806]
  MoveL 257 to (-162.16, 1350, -0.5) mm, rotated rx -180 ry 0 rz 90 deg; joints [-29.753, -95.954, 143.955, 69.95, 19.418, -92.797]
  MoveL 258 to (-162.16, 1350, 50) mm, rotated rx 180 ry 0 rz 90 deg; joints [-29.753, -99.244, 143.032, 59.637, 21.22, -81.806]
  MoveL 259 to (-162.16, 1400, 50) mm, rotated rx -180 ry 0 rz 90 deg; joints [-31.234, -101.939, 145.051, 58.55, 22.49, -81.731]
  MoveL 260 to (-162.16, 1400, -0.5) mm, rotated rx -180 ry 0 rz 90 deg; joints [-31.234, -98.499, 146.025, 68.602, 20.517, -92.529]
  MoveL 261 to (-162.16, 1400, 50) mm, rotated rx -180 ry 0 rz 90 deg; joints [-31.234, -101.939, 145.051, 58.55, 22.49, -81.731]
  MoveL 262 to (-237.84, 50, 50) mm, rotated rx 180 ry 0 rz 90 deg; joints [-11.004, -46.16, 71.7, 15.443, 26.817, -22.443]
  MoveL 263 to (-237.84, 50, -0.5) mm, rotated rx 180 ry 0 rz 90 deg; joints [-11.004, -44.914, 72.245, 16.453, 25.096, -23.567]
  MoveL 264 to (-237.84, 50, 50) mm, rotated rx 180 ry 0 rz 90 deg; joints [-11.004, -46.16, 71.7, 15.443, 26.817, -22.443]
  MoveL 265 to (-237.84, 100, 50) mm, rotated rx 180 ry 0 rz 90 deg; joints [-11.257, -48.381, 75.562, 16.704, 25.304, -23.972]
  MoveL 266 to (-237.84, 100, -0.5) mm, rotated rx 180 ry 0 rz 90 deg; joints [-11.257, -47.092, 76.098, 17.899, 23.561, -25.284]
  MoveL 267 to (-237.84, 100, 50) mm, rotated rx 180 ry 0 rz 90 deg; joints [-11.257, -48.381, 75.562, 16.704, 25.304, -23.972]
  MoveL 268 to (-237.84, 150, 50) mm, rotated rx -180 ry 0 rz 90 deg; joints [-11.522, -50.535, 79.263, 18.077, 23.897, -25.619]
  MoveL 269 to (-237.84, 150, -0.5) mm, rotated rx 180 ry 0 rz 90 deg; joints [-11.522, -49.201, 79.793, 19.49, 22.133, -27.153]
  MoveL 270 to (-237.84, 150, 50) mm, rotated rx -180 ry 0 rz 90 deg; joints [-11.522, -50.535, 79.263, 18.077, 23.897, -25.619]
  MoveL 271 to (-237.84, 200, 50) mm, rotated rx -180 ry 0 rz 90 deg; joints [-11.799, -52.633, 82.824, 19.572, 22.59, -27.394]
  MoveL 272 to (-237.84, 200, -0.5) mm, rotated rx -180 ry 0 rz 90 deg; joints [-11.799, -51.254, 83.349, 21.241, 20.805, -29.19]
  MoveL 273 to (-237.84, 200, 50) mm, rotated rx -180 ry 0 rz 90 deg; joints [-11.799, -52.633, 82.824, 19.572, 22.59, -27.394]
  MoveL 274 to (-237.84, 250, 50) mm, rotated rx 180 ry 0 rz 90 deg; joints [-12.09, -54.685, 86.261, 21.198, 21.378, -29.308]
  MoveL 275 to (-237.84, 250, -0.5) mm, rotated rx 180 ry 0 rz 90 deg; joints [-12.09, -53.259, 86.785, 23.17, 19.572, -31.412]
  MoveL 276 to (-237.84, 250, 50) mm, rotated rx 180 ry 0 rz 90 deg; joints [-12.09, -54.685, 86.261, 21.198, 21.378, -29.308]
  MoveL 277 to (-237.84, 300, 50) mm, rotated rx 180 ry 0 rz 90 deg; joints [-12.395, -56.698, 89.589, 22.964, 20.257, -31.371]
  MoveL 278 to (-237.84, 300, -0.5) mm, rotated rx 180 ry 0 rz 90 deg; joints [-12.395, -55.224, 90.113, 25.29, 18.433, -33.836]
  MoveL 279 to (-237.84, 300, 50) mm, rotated rx 180 ry 0 rz 90 deg; joints [-12.395, -56.698, 89.589, 22.964, 20.257, -31.371]
  MoveL 280 to (-237.84, 350, 50) mm, rotated rx 180 ry 0 rz 90 deg; joints [-12.715, -58.682, 92.82, 24.876, 19.225, -33.591]
  MoveL 281 to (-237.84, 350, -0.5) mm, rotated rx 180 ry 0 rz 90 deg; joints [-12.715, -57.158, 93.345, 27.617, 17.386, -36.477]
  MoveL 282 to (-237.84, 350, 50) mm, rotated rx 180 ry 0 rz 90 deg; joints [-12.715, -58.682, 92.82, 24.876, 19.225, -33.591]
  MoveL 283 to (-237.84, 400, 50) mm, rotated rx -180 ry 0 rz 90 deg; joints [-13.053, -60.641, 95.961, 26.94, 18.283, -35.973]
  MoveL 284 to (-237.84, 400, -0.5) mm, rotated rx 180 ry 0 rz 90 deg; joints [-13.053, -59.065, 96.49, 30.16, 16.433, -39.346]
  MoveL 285 to (-237.84, 400, 50) mm, rotated rx -180 ry 0 rz 90 deg; joints [-13.053, -60.641, 95.961, 26.94, 18.283, -35.973]
  MoveL 286 to (-237.84, 450, 50) mm, rotated rx -180 ry 0 rz 90 deg; joints [-13.408, -62.583, 99.022, 29.155, 17.43, -38.519]
  MoveL 287 to (-237.84, 450, -0.5) mm, rotated rx 180 ry 0 rz 90 deg; joints [-13.408, -60.952, 99.556, 32.924, 15.574, -42.449]
  MoveL 288 to (-237.84, 450, 50) mm, rotated rx -180 ry 0 rz 90 deg; joints [-13.408, -62.583, 99.022, 29.155, 17.43, -38.519]
  MoveL 289 to (-237.84, 500, 50) mm, rotated rx 180 ry 0 rz 90 deg; joints [-13.783, -64.512, 102.01, 31.515, 16.668, -41.223]
  MoveL 290 to (-237.84, 500, -0.5) mm, rotated rx 180 ry 0 rz 90 deg; joints [-13.783, -62.824, 102.55, 35.904, 14.813, -45.783]
  MoveL 291 to (-237.84, 500, 50) mm, rotated rx 180 ry 0 rz 90 deg; joints [-13.783, -64.512, 102.01, 31.515, 16.668, -41.223]
  MoveL 292 to (-237.84, 550, 50) mm, rotated rx 180 ry 0 rz 90 deg; joints [-14.179, -66.435, 104.929, 34.008, 15.998, -44.075]
  MoveL 293 to (-237.84, 550, -0.5) mm, rotated rx 180 ry 0 rz 90 deg; joints [-14.179, -64.686, 105.477, 39.087, 14.152, -49.334]
  MoveL 294 to (-237.84, 550, 50) mm, rotated rx 180 ry 0 rz 90 deg; joints [-14.179, -66.435, 104.929, 34.008, 15.998, -44.075]
  MoveL 295 to (-237.84, 600, 50) mm, rotated rx -180 ry 0 rz 90 deg; joints [-14.598, -68.356, 107.786, 36.613, 15.423, -47.055]
  MoveL 296 to (-237.84, 600, -0.5) mm, rotated rx -180 ry 0 rz 90 deg; joints [-14.598, -66.544, 108.343, 42.443, 13.593, -53.075]
  MoveL 297 to (-237.84, 600, 50) mm, rotated rx -180 ry 0 rz 90 deg; joints [-14.598, -68.356, 107.786, 36.613, 15.423, -47.055]
  MoveL 298 to (-237.84, 650, 50) mm, rotated rx -180 ry 0 rz 90 deg; joints [-15.042, -70.28, 110.583, 39.298, 14.944, -50.132]
  MoveL 299 to (-237.84, 650, -0.5) mm, rotated rx 180 ry 0 rz 90 deg; joints [-15.042, -68.401, 111.151, 45.926, 13.14, -56.962]
  MoveL 300 to (-237.84, 650, 50) mm, rotated rx -180 ry 0 rz 90 deg; joints [-15.042, -70.28, 110.583, 39.298, 14.944, -50.132]
  MoveL 301 to (-237.84, 700, 50) mm, rotated rx -180 ry 0 rz 90 deg; joints [-15.513, -72.213, 113.326, 42.023, 14.562, -53.267]
  MoveL 302 to (-237.84, 700, -0.5) mm, rotated rx 180 ry 0 rz 90 deg; joints [-15.513, -70.263, 113.906, 49.475, 12.793, -60.935]
  MoveL 303 to (-237.84, 700, 50) mm, rotated rx -180 ry 0 rz 90 deg; joints [-15.513, -72.213, 113.326, 42.023, 14.562, -53.267]
  MoveL 304 to (-237.84, 750, 50) mm, rotated rx 180 ry 0 rz 90 deg; joints [-16.013, -74.16, 116.016, 44.736, 14.28, -56.411]
  MoveL 305 to (-237.84, 750, -0.5) mm, rotated rx 180 ry 0 rz 90 deg; joints [-16.013, -72.136, 116.611, 53.016, 12.553, -64.921]
  MoveL 306 to (-237.84, 750, 50) mm, rotated rx 180 ry 0 rz 90 deg; joints [-16.013, -74.16, 116.016, 44.736, 14.28, -56.411]
  MoveL 307 to (-237.84, 800, 50) mm, rotated rx -180 ry 0 rz 90 deg; joints [-16.547, -76.128, 118.657, 47.381, 14.097, -59.508]
  MoveL 308 to (-237.84, 800, -0.5) mm, rotated rx 180 ry 0 rz 90 deg; joints [-16.547, -74.023, 119.267, 56.461, 12.417, -68.835]
  MoveL 309 to (-237.84, 800, 50) mm, rotated rx -180 ry 0 rz 90 deg; joints [-16.547, -76.128, 118.657, 47.381, 14.097, -59.508]
  MoveL 310 to (-237.84, 850, 50) mm, rotated rx 180 ry 0 rz 90 deg; joints [-17.115, -78.121, 121.25, 49.893, 14.014, -62.496]
  MoveL 311 to (-237.84, 850, -0.5) mm, rotated rx 180 ry 0 rz 90 deg; joints [-17.115, -75.932, 121.878, 59.723, 12.384, -72.59]
  MoveL 312 to (-237.84, 850, 50) mm, rotated rx 180 ry 0 rz 90 deg; joints [-17.115, -78.121, 121.25, 49.893, 14.014, -62.496]
  MoveL 313 to (-237.84, 900, 50) mm, rotated rx -180 ry 0 rz 90 deg; joints [-17.723, -80.148, 123.797, 52.209, 14.03, -65.313]
  MoveL 314 to (-237.84, 900, -0.5) mm, rotated rx 180 ry 0 rz 90 deg; joints [-17.723, -77.869, 124.445, 62.714, 12.449, -76.104]
  MoveL 315 to (-237.84, 900, 50) mm, rotated rx -180 ry 0 rz 90 deg; joints [-17.723, -80.148, 123.797, 52.209, 14.03, -65.313]
  MoveL 316 to (-237.84, 950, 50) mm, rotated rx -180 ry 0 rz 90 deg; joints [-18.375, -82.215, 126.3, 54.267, 14.145, -67.901]
  MoveL 317 to (-237.84, 950, -0.5) mm, rotated rx -180 ry 0 rz 90 deg; joints [-18.375, -79.839, 126.97, 65.359, 12.607, -79.299]
  MoveL 318 to (-237.84, 950, 50) mm, rotated rx -180 ry 0 rz 90 deg; joints [-18.375, -82.215, 126.3, 54.267, 14.145, -67.901]
  MoveL 319 to (-237.84, 1000, 50) mm, rotated rx -180 ry 0 rz 90 deg; joints [-19.074, -84.331, 128.758, 56.014, 14.36, -70.207]
  MoveL 320 to (-237.84, 1000, -0.5) mm, rotated rx -180 ry 0 rz 90 deg; joints [-19.074, -81.852, 129.453, 67.591, 12.853, -82.115]
  MoveL 321 to (-237.84, 1000, 50) mm, rotated rx -180 ry 0 rz 90 deg; joints [-19.074, -84.331, 128.758, 56.014, 14.36, -70.207]
  MoveL 322 to (-237.84, 1050, 50) mm, rotated rx 180 ry 0 rz 90 deg; joints [-19.826, -86.504, 131.173, 57.403, 14.676, -72.186]
  MoveL 323 to (-237.84, 1050, -0.5) mm, rotated rx 180 ry 0 rz 90 deg; joints [-19.826, -83.915, 131.895, 69.36, 13.184, -84.502]
  MoveL 324 to (-237.84, 1050, 50) mm, rotated rx 180 ry 0 rz 90 deg; joints [-19.826, -86.504, 131.173, 57.403, 14.676, -72.186]
  MoveL 325 to (-237.84, 1100, 50) mm, rotated rx 180 ry 0 rz 90 deg; joints [-20.637, -88.745, 133.544, 58.397, 15.095, -73.806]
  MoveL 326 to (-237.84, 1100, -0.5) mm, rotated rx 180 ry 0 rz 90 deg; joints [-20.637, -86.038, 134.296, 70.63, 13.598, -86.428]
  MoveL 327 to (-237.84, 1100, 50) mm, rotated rx 180 ry 0 rz 90 deg; joints [-20.637, -88.745, 133.544, 58.397, 15.095, -73.806]
  MoveL 328 to (-237.84, 1150, 50) mm, rotated rx -180 ry 0 rz 90 deg; joints [-21.514, -91.065, 135.87, 58.973, 15.624, -75.045]
  MoveL 329 to (-237.84, 1150, -0.5) mm, rotated rx 180 ry 0 rz 90 deg; joints [-21.514, -88.234, 136.656, 71.375, 14.096, -87.871]
  MoveL 330 to (-237.84, 1150, 50) mm, rotated rx -180 ry 0 rz 90 deg; joints [-21.514, -91.065, 135.87, 58.973, 15.624, -75.045]
  MoveL 331 to (-237.84, 1200, 50) mm, rotated rx 180 ry 0 rz 90 deg; joints [-22.465, -93.479, 138.15, 59.119, 16.272, -75.892]
  MoveL 332 to (-237.84, 1200, -0.5) mm, rotated rx 180 ry 0 rz 90 deg; joints [-22.465, -90.514, 138.973, 71.583, 14.682, -88.82]
  MoveL 333 to (-237.84, 1200, 50) mm, rotated rx 180 ry 0 rz 90 deg; joints [-22.465, -93.479, 138.15, 59.119, 16.272, -75.892]
  MoveL 334 to (-237.84, 1250, 50) mm, rotated rx 180 ry 0 rz 90 deg; joints [-23.499, -96.001, 140.382, 58.834, 17.053, -76.351]
  MoveL 335 to (-237.84, 1250, -0.5) mm, rotated rx 180 ry 0 rz 90 deg; joints [-23.499, -92.894, 141.247, 71.25, 15.367, -89.276]
  MoveL 336 to (-237.84, 1250, 50) mm, rotated rx 180 ry 0 rz 90 deg; joints [-23.499, -96.001, 140.382, 58.834, 17.053, -76.351]
  MoveL 337 to (-237.84, 1300, 50) mm, rotated rx 180 ry 0 rz 90 deg; joints [-24.627, -98.648, 142.563, 58.129, 17.987, -76.436]
  MoveL 338 to (-237.84, 1300, -0.5) mm, rotated rx -180 ry 0 rz 90 deg; joints [-24.627, -95.392, 143.475, 70.381, 16.165, -89.246]
  MoveL 339 to (-237.84, 1300, 50) mm, rotated rx 180 ry 0 rz 90 deg; joints [-24.627, -98.648, 142.563, 58.129, 17.987, -76.436]
  MoveL 340 to (-237.84, 1350, 50) mm, rotated rx -180 ry 0 rz 90 deg; joints [-25.86, -101.441, 144.69, 57.031, 19.098, -76.175]
  MoveL 341 to (-237.84, 1350, -0.5) mm, rotated rx 180 ry 0 rz 90 deg; joints [-25.86, -98.028, 145.654, 68.993, 17.1, -88.752]
  MoveL 342 to (-237.84, 1350, 50) mm, rotated rx -180 ry 0 rz 90 deg; joints [-25.86, -101.441, 144.69, 57.031, 19.098, -76.175]
  MoveL 343 to (-313.52, 50, 50) mm, rotated rx 180 ry 0 rz 90 deg; joints [-9.068, -46.764, 72.756, 13.101, 25.95, -18.889]
  MoveL 344 to (-313.52, 50, -0.5) mm, rotated rx 180 ry 0 rz 90 deg; joints [-9.068, -45.507, 73.298, 14.001, 24.201, -19.884]
  MoveL 345 to (-313.52, 50, 50) mm, rotated rx 180 ry 0 rz 90 deg; joints [-9.068, -46.764, 72.756, 13.101, 25.95, -18.889]
  MoveL 346 to (-313.52, 100, 50) mm, rotated rx 180 ry 0 rz 90 deg; joints [-9.278, -48.98, 76.596, 14.209, 24.416, -20.218]
  MoveL 347 to (-313.52, 100, -0.5) mm, rotated rx 180 ry 0 rz 90 deg; joints [-9.278, -47.679, 77.129, 15.282, 22.641, -21.388]
  MoveL 348 to (-313.52, 100, 50) mm, rotated rx 180 ry 0 rz 90 deg; joints [-9.278, -48.98, 76.596, 14.209, 24.416, -20.218]
  MoveL 349 to (-313.52, 150, 50) mm, rotated rx 180 ry 0 rz 90 deg; joints [-9.498, -51.132, 80.28, 15.424, 22.984, -21.659]
  MoveL 350 to (-313.52, 150, -0.5) mm, rotated rx -180 ry 0 rz 90 deg; joints [-9.498, -49.785, 80.808, 16.702, 21.182, -23.039]
  MoveL 351 to (-313.52, 150, 50) mm, rotated rx 180 ry 0 rz 90 deg; joints [-9.498, -51.132, 80.28, 15.424, 22.984, -21.659]
  MoveL 352 to (-313.52, 200, 50) mm, rotated rx 180 ry 0 rz 90 deg; joints [-9.728, -53.23, 83.829, 16.756, 21.645, -23.224]
  MoveL 353 to (-313.52, 200, -0.5) mm, rotated rx 180 ry 0 rz 90 deg; joints [-9.728, -51.837, 84.354, 18.281, 19.817, -24.854]
  MoveL 354 to (-313.52, 200, 50) mm, rotated rx 180 ry 0 rz 90 deg; joints [-9.728, -53.23, 83.829, 16.756, 21.645, -23.224]
  MoveL 355 to (-313.52, 250, 50) mm, rotated rx 180 ry 0 rz 90 deg; joints [-9.97, -55.285, 87.258, 18.219, 20.396, -24.925]
  MoveL 356 to (-313.52, 250, -0.5) mm, rotated rx 180 ry 0 rz 90 deg; joints [-9.97, -53.845, 87.782, 20.039, 18.541, -26.856]
  MoveL 357 to (-313.52, 250, 50) mm, rotated rx 180 ry 0 rz 90 deg; joints [-9.97, -55.285, 87.258, 18.219, 20.396, -24.925]
  MoveL 358 to (-313.52, 300, 50) mm, rotated rx -180 ry 0 rz 90 deg; joints [-10.225, -57.304, 90.581, 19.823, 19.233, -26.775]
  MoveL 359 to (-313.52, 300, -0.5) mm, rotated rx 180 ry 0 rz 90 deg; joints [-10.225, -55.815, 91.106, 21.997, 17.352, -29.065]
  MoveL 360 to (-313.52, 300, 50) mm, rotated rx -180 ry 0 rz 90 deg; joints [-10.225, -57.304, 90.581, 19.823, 19.233, -26.775]
  MoveL 361 to (-313.52, 350, 50) mm, rotated rx 180 ry 0 rz 90 deg; joints [-10.492, -59.296, 93.81, 21.579, 18.155, -28.786]
  MoveL 362 to (-313.52, 350, -0.5) mm, rotated rx -180 ry 0 rz 90 deg; joints [-10.492, -57.756, 94.336, 24.174, 16.25, -31.503]
  MoveL 363 to (-313.52, 350, 50) mm, rotated rx 180 ry 0 rz 90 deg; joints [-10.492, -59.296, 93.81, 21.579, 18.155, -28.786]
  MoveL 364 to (-313.52, 400, 50) mm, rotated rx 180 ry 0 rz 90 deg; joints [-10.773, -61.266, 96.952, 23.497, 17.16, -30.969]
  MoveL 365 to (-313.52, 400, -0.5) mm, rotated rx 180 ry 0 rz 90 deg; joints [-10.773, -59.672, 97.482, 26.593, 15.235, -34.192]
  MoveL 366 to (-313.52, 400, 50) mm, rotated rx 180 ry 0 rz 90 deg; joints [-10.773, -61.266, 96.952, 23.497, 17.16, -30.969]
  MoveL 367 to (-313.52, 450, 50) mm, rotated rx -180 ry 0 rz 90 deg; joints [-11.07, -63.221, 100.016, 25.582, 16.25, -33.329]
  MoveL 368 to (-313.52, 450, -0.5) mm, rotated rx 180 ry 0 rz 90 deg; joints [-11.07, -61.571, 100.552, 29.267, 14.31, -37.149]
  MoveL 369 to (-313.52, 450, 50) mm, rotated rx -180 ry 0 rz 90 deg; joints [-11.07, -63.221, 100.016, 25.582, 16.25, -33.329]
  MoveL 370 to (-313.52, 500, 50) mm, rotated rx 180 ry 0 rz 90 deg; joints [-11.383, -65.166, 103.009, 27.837, 15.426, -35.87]
  MoveL 371 to (-313.52, 500, -0.5) mm, rotated rx 180 ry 0 rz 90 deg; joints [-11.383, -63.458, 103.551, 32.209, 13.476, -40.384]
  MoveL 372 to (-313.52, 500, 50) mm, rotated rx 180 ry 0 rz 90 deg; joints [-11.383, -65.166, 103.009, 27.837, 15.426, -35.87]
  MoveL 373 to (-313.52, 550, 50) mm, rotated rx 180 ry 0 rz 90 deg; joints [-11.715, -67.107, 105.936, 30.255, 14.69, -38.588]
  MoveL 374 to (-313.52, 550, -0.5) mm, rotated rx -180 ry 0 rz 90 deg; joints [-11.715, -65.337, 106.487, 35.415, 12.738, -43.898]
  MoveL 375 to (-313.52, 550, 50) mm, rotated rx 180 ry 0 rz 90 deg; joints [-11.715, -67.107, 105.936, 30.255, 14.69, -38.588]
  MoveL 376 to (-313.52, 600, 50) mm, rotated rx 180 ry 0 rz 90 deg; joints [-12.066, -69.049, 108.802, 32.824, 14.045, -41.468]
  MoveL 377 to (-313.52, 600, -0.5) mm, rotated rx 180 ry 0 rz 90 deg; joints [-12.066, -67.214, 109.363, 38.871, 12.1, -47.675]
  MoveL 378 to (-313.52, 600, 50) mm, rotated rx 180 ry 0 rz 90 deg; joints [-12.066, -69.049, 108.802, 32.824, 14.045, -41.468]
  MoveL 379 to (-313.52, 650, 50) mm, rotated rx -180 ry 0 rz 90 deg; joints [-12.438, -70.998, 111.611, 35.515, 13.493, -44.487]
  MoveL 380 to (-313.52, 650, -0.5) mm, rotated rx -180 ry 0 rz 90 deg; joints [-12.438, -69.094, 112.184, 42.539, 11.565, -51.681]
  MoveL 381 to (-313.52, 650, 50) mm, rotated rx -180 ry 0 rz 90 deg; joints [-12.438, -70.998, 111.611, 35.515, 13.493, -44.487]
  MoveL 382 to (-313.52, 700, 50) mm, rotated rx -180 ry 0 rz 90 deg; joints [-12.833, -72.96, 114.367, 38.292, 13.037, -47.606]
  MoveL 383 to (-313.52, 700, -0.5) mm, rotated rx 180 ry 0 rz 90 deg; joints [-12.833, -70.983, 114.953, 46.36, 11.137, -55.855]
  MoveL 384 to (-313.52, 700, 50) mm, rotated rx -180 ry 0 rz 90 deg; joints [-12.833, -72.96, 114.367, 38.292, 13.037, -47.606]
  MoveL 385 to (-313.52, 750, 50) mm, rotated rx -180 ry 0 rz 90 deg; joints [-13.254, -74.941, 117.073, 41.101, 12.679, -50.775]
  MoveL 386 to (-313.52, 750, -0.5) mm, rotated rx -180 ry 0 rz 90 deg; joints [-13.254, -72.885, 117.674, 50.25, 10.817, -60.117]
  MoveL 387 to (-313.52, 750, 50) mm, rotated rx -180 ry 0 rz 90 deg; joints [-13.254, -74.941, 117.073, 41.101, 12.679, -50.775]
  MoveL 388 to (-313.52, 800, 50) mm, rotated rx -180 ry 0 rz 90 deg; joints [-13.703, -76.946, 119.732, 43.877, 12.421, -53.93]
  MoveL 389 to (-313.52, 800, -0.5) mm, rotated rx -180 ry 0 rz 90 deg; joints [-13.703, -74.808, 120.349, 54.102, 10.605, -64.363]
  MoveL 390 to (-313.52, 800, 50) mm, rotated rx -180 ry 0 rz 90 deg; joints [-13.703, -76.946, 119.732, 43.877, 12.421, -53.93]
  MoveL 391 to (-313.52, 850, 50) mm, rotated rx 180 ry 0 rz 90 deg; joints [-14.183, -78.984, 122.345, 46.546, 12.264, -56.997]
  MoveL 392 to (-313.52, 850, -0.5) mm, rotated rx -180 ry 0 rz 90 deg; joints [-14.183, -76.757, 122.981, 57.801, 10.499, -68.475]
  MoveL 393 to (-313.52, 850, 50) mm, rotated rx 180 ry 0 rz 90 deg; joints [-14.183, -78.984, 122.345, 46.546, 12.264, -56.997]
  MoveL 394 to (-313.52, 900, 50) mm, rotated rx -180 ry 0 rz 90 deg; joints [-14.697, -81.061, 124.914, 49.026, 12.209, -59.898]
  MoveL 395 to (-313.52, 900, -0.5) mm, rotated rx -180 ry 0 rz 90 deg; joints [-14.697, -78.739, 125.572, 61.224, 10.496, -72.336]
  MoveL 396 to (-313.52, 900, 50) mm, rotated rx -180 ry 0 rz 90 deg; joints [-14.697, -81.061, 124.914, 49.026, 12.209, -59.898]
  MoveL 397 to (-313.52, 950, 50) mm, rotated rx 180 ry 0 rz 90 deg; joints [-15.249, -83.186, 127.441, 51.237, 12.256, -62.552]
  MoveL 398 to (-313.52, 950, -0.5) mm, rotated rx -180 ry 0 rz 90 deg; joints [-15.249, -80.763, 128.122, 64.258, 10.589, -75.833]
  MoveL 399 to (-313.52, 950, 50) mm, rotated rx 180 ry 0 rz 90 deg; joints [-15.249, -83.186, 127.441, 51.237, 12.256, -62.552]
  MoveL 400 to (-313.52, 1000, 50) mm, rotated rx 180 ry 0 rz 90 deg; joints [-15.843, -85.368, 129.926, 53.103, 12.406, -64.888]
  MoveL 401 to (-313.52, 1000, -0.5) mm, rotated rx -180 ry 0 rz 90 deg; joints [-15.843, -82.838, 130.633, 66.807, 10.773, -78.873]
  MoveL 402 to (-313.52, 1000, 50) mm, rotated rx 180 ry 0 rz 90 deg; joints [-15.843, -85.368, 129.926, 53.103, 12.406, -64.888]
  MoveL 403 to (-313.52, 1050, 50) mm, rotated rx 180 ry 0 rz 90 deg; joints [-16.483, -87.62, 132.369, 54.56, 12.66, -66.841]
  MoveL 404 to (-313.52, 1050, -0.5) mm, rotated rx -180 ry 0 rz 90 deg; joints [-16.483, -84.973, 133.106, 68.793, 11.042, -81.38]
  MoveL 405 to (-313.52, 1050, 50) mm, rotated rx 180 ry 0 rz 90 deg; joints [-16.483, -87.62, 132.369, 54.56, 12.66, -66.841]
  MoveL 406 to (-313.52, 1100, 50) mm, rotated rx -180 ry 0 rz 90 deg; joints [-17.176, -89.952, 134.771, 55.555, 13.024, -68.363]
  MoveL 407 to (-313.52, 1100, -0.5) mm, rotated rx 180 ry 0 rz 90 deg; joints [-17.176, -87.181, 135.54, 70.159, 11.395, -83.3]
  MoveL 408 to (-313.52, 1100, 50) mm, rotated rx -180 ry 0 rz 90 deg; joints [-17.176, -89.952, 134.771, 55.555, 13.024, -68.363]
  MoveL 409 to (-313.52, 1150, 50) mm, rotated rx -180 ry 0 rz 90 deg; joints [-17.928, -92.381, 137.13, 56.055, 13.504, -69.421]
  MoveL 410 to (-313.52, 1150, -0.5) mm, rotated rx -180 ry 0 rz 90 deg; joints [-17.928, -89.477, 137.936, 70.868, 11.832, -84.597]
  MoveL 411 to (-313.52, 1150, 50) mm, rotated rx -180 ry 0 rz 90 deg; joints [-17.928, -92.381, 137.13, 56.055, 13.504, -69.421]
  MoveL 412 to (-313.52, 1200, 50) mm, rotated rx 180 ry 0 rz 90 deg; joints [-18.746, -94.922, 139.446, 56.042, 14.113, -69.999]
  MoveL 413 to (-313.52, 1200, -0.5) mm, rotated rx 180 ry 0 rz 90 deg; joints [-18.746, -91.876, 140.293, 70.898, 12.359, -85.253]
  MoveL 414 to (-313.52, 1200, 50) mm, rotated rx 180 ry 0 rz 90 deg; joints [-18.746, -94.922, 139.446, 56.042, 14.113, -69.999]
  MoveL 415 to (-313.52, 1250, 50) mm, rotated rx 180 ry 0 rz 90 deg; joints [-19.639, -97.596, 141.716, 55.516, 14.868, -70.1]
  MoveL 416 to (-313.52, 1250, -0.5) mm, rotated rx 180 ry 0 rz 90 deg; joints [-19.639, -94.399, 142.609, 70.242, 12.988, -85.264]
  MoveL 417 to (-313.52, 1250, 50) mm, rotated rx 180 ry 0 rz 90 deg; joints [-19.639, -97.596, 141.716, 55.516, 14.868, -70.1]
  MoveL 418 to (-313.52, 1300, 50) mm, rotated rx -180 ry 0 rz 90 deg; joints [-20.617, -100.425, 143.937, 54.498, 15.796, -69.747]
  MoveL 419 to (-313.52, 1300, -0.5) mm, rotated rx 180 ry 0 rz 90 deg; joints [-20.617, -97.069, 144.882, 68.909, 13.74, -84.642]
  MoveL 420 to (-313.52, 1300, 50) mm, rotated rx -180 ry 0 rz 90 deg; joints [-20.617, -100.425, 143.937, 54.498, 15.796, -69.747]
  MoveL 421 to (-389.2, 50, 50) mm, rotated rx 180 ry 0 rz 90 deg; joints [-7.11, -47.248, 73.598, 10.526, 25.239, -15.078]
  MoveL 422 to (-389.2, 50, -0.5) mm, rotated rx 180 ry 0 rz 90 deg; joints [-7.11, -45.982, 74.138, 11.281, 23.465, -15.906]
  MoveL 423 to (-389.2, 50, 50) mm, rotated rx 180 ry 0 rz 90 deg; joints [-7.11, -47.248, 73.598, 10.526, 25.239, -15.078]
  MoveL 424 to (-389.2, 100, 50) mm, rotated rx 180 ry 0 rz 90 deg; joints [-7.276, -49.46, 77.422, 11.444, 23.685, -16.169]
  MoveL 425 to (-389.2, 100, -0.5) mm, rotated rx 180 ry 0 rz 90 deg; joints [-7.276, -48.149, 77.954, 12.349, 21.881, -17.15]
  MoveL 426 to (-389.2, 100, 50) mm, rotated rx 180 ry 0 rz 90 deg; joints [-7.276, -49.46, 77.422, 11.444, 23.685, -16.169]
  MoveL 427 to (-389.2, 150, 50) mm, rotated rx 180 ry 0 rz 90 deg; joints [-7.45, -51.611, 81.094, 12.457, 22.228, -17.359]
  MoveL 428 to (-389.2, 150, -0.5) mm, rotated rx 180 ry 0 rz 90 deg; joints [-7.45, -50.254, 81.621, 13.543, 20.392, -18.525]
  MoveL 429 to (-389.2, 150, 50) mm, rotated rx 180 ry 0 rz 90 deg; joints [-7.45, -51.611, 81.094, 12.457, 22.228, -17.359]
  MoveL 430 to (-389.2, 200, 50) mm, rotated rx 180 ry 0 rz 90 deg; joints [-7.632, -53.71, 84.634, 13.575, 20.86, -18.66]
  MoveL 431 to (-389.2, 200, -0.5) mm, rotated rx -180 ry 0 rz 90 deg; joints [-7.632, -52.306, 85.158, 14.883, 18.991, -20.051]
  MoveL 432 to (-389.2, 200, 50) mm, rotated rx 180 ry 0 rz 90 deg; joints [-7.632, -53.71, 84.634, 13.575, 20.86, -18.66]
  MoveL 433 to (-389.2, 250, 50) mm, rotated rx 180 ry 0 rz 90 deg; joints [-7.823, -55.768, 88.057, 14.813, 19.576, -20.086]
  MoveL 434 to (-389.2, 250, -0.5) mm, rotated rx 180 ry 0 rz 90 deg; joints [-7.823, -54.316, 88.581, 16.39, 17.673, -21.75]
  MoveL 435 to (-389.2, 250, 50) mm, rotated rx 180 ry 0 rz 90 deg; joints [-7.823, -55.768, 88.057, 14.813, 19.576, -20.086]
  MoveL 436 to (-389.2, 300, 50) mm, rotated rx -180 ry 0 rz 90 deg; joints [-8.024, -57.793, 91.377, 16.183, 18.372, -21.651]
  MoveL 437 to (-389.2, 300, -0.5) mm, rotated rx -180 ry 0 rz 90 deg; joints [-8.024, -56.291, 91.902, 18.088, 16.436, -23.647]
  MoveL 438 to (-389.2, 300, 50) mm, rotated rx -180 ry 0 rz 90 deg; joints [-8.024, -57.793, 91.377, 16.183, 18.372, -21.651]
  MoveL 439 to (-389.2, 350, 50) mm, rotated rx 180 ry 0 rz 90 deg; joints [-8.236, -59.791, 94.605, 17.7, 17.248, -23.368]
  MoveL 440 to (-389.2, 350, -0.5) mm, rotated rx 180 ry 0 rz 90 deg; joints [-8.236, -58.238, 95.132, 20.005, 15.279, -25.769]
  MoveL 441 to (-389.2, 350, 50) mm, rotated rx 180 ry 0 rz 90 deg; joints [-8.236, -59.791, 94.605, 17.7, 17.248, -23.368]
  MoveL 442 to (-389.2, 400, 50) mm, rotated rx 180 ry 0 rz 90 deg; joints [-8.459, -61.771, 97.748, 19.376, 16.202, -25.253]
  MoveL 443 to (-389.2, 400, -0.5) mm, rotated rx -180 ry 0 rz 90 deg; joints [-8.459, -60.163, 98.279, 22.169, 14.201, -28.147]
  MoveL 444 to (-389.2, 400, 50) mm, rotated rx 180 ry 0 rz 90 deg; joints [-8.459, -61.771, 97.748, 19.376, 16.202, -25.253]
  MoveL 445 to (-389.2, 450, 50) mm, rotated rx -180 ry 0 rz 90 deg; joints [-8.694, -63.737, 100.815, 21.223, 15.235, -27.318]
  MoveL 446 to (-389.2, 450, -0.5) mm, rotated rx -180 ry 0 rz 90 deg; joints [-8.694, -62.072, 101.352, 24.608, 13.205, -30.809]
  MoveL 447 to (-389.2, 450, 50) mm, rotated rx -180 ry 0 rz 90 deg; joints [-8.694, -63.737, 100.815, 21.223, 15.235, -27.318]
  MoveL 448 to (-389.2, 500, 50) mm, rotated rx 180 ry 0 rz 90 deg; joints [-8.942, -65.695, 103.813, 23.252, 14.347, -29.572]
  MoveL 449 to (-389.2, 500, -0.5) mm, rotated rx -180 ry 0 rz 90 deg; joints [-8.942, -63.97, 104.357, 27.35, 12.294, -33.783]
  MoveL 450 to (-389.2, 500, 50) mm, rotated rx 180 ry 0 rz 90 deg; joints [-8.942, -65.695, 103.813, 23.252, 14.347, -29.572]
  MoveL 451 to (-389.2, 550, 50) mm, rotated rx 180 ry 0 rz 90 deg; joints [-9.206, -67.652, 106.746, 25.465, 13.542, -32.022]
  MoveL 452 to (-389.2, 550, -0.5) mm, rotated rx 180 ry 0 rz 90 deg; joints [-9.206, -65.864, 107.3, 30.413, 11.471, -37.089]
  MoveL 453 to (-389.2, 550, 50) mm, rotated rx 180 ry 0 rz 90 deg; joints [-9.206, -67.652, 106.746, 25.465, 13.542, -32.022]
  MoveL 454 to (-389.2, 600, 50) mm, rotated rx 180 ry 0 rz 90 deg; joints [-9.484, -69.613, 109.621, 27.858, 12.822, -34.662]
  MoveL 455 to (-389.2, 600, -0.5) mm, rotated rx -180 ry 0 rz 90 deg; joints [-9.484, -67.758, 110.185, 33.806, 10.742, -40.737]
  MoveL 456 to (-389.2, 600, 50) mm, rotated rx 180 ry 0 rz 90 deg; joints [-9.484, -69.613, 109.621, 27.858, 12.822, -34.662]
  MoveL 457 to (-389.2, 650, 50) mm, rotated rx -180 ry 0 rz 90 deg; joints [-9.781, -71.583, 112.44, 30.417, 12.19, -37.48]
  MoveL 458 to (-389.2, 650, -0.5) mm, rotated rx 180 ry 0 rz 90 deg; joints [-9.781, -69.657, 113.016, 37.515, 10.111, -44.713]
  MoveL 459 to (-389.2, 650, 50) mm, rotated rx -180 ry 0 rz 90 deg; joints [-9.781, -71.583, 112.44, 30.417, 12.19, -37.48]
  MoveL 460 to (-389.2, 700, 50) mm, rotated rx 180 ry 0 rz 90 deg; joints [-10.096, -73.569, 115.208, 33.113, 11.65, -40.448]
  MoveL 461 to (-389.2, 700, -0.5) mm, rotated rx -180 ry 0 rz 90 deg; joints [-10.096, -71.568, 115.798, 41.501, 9.583, -48.979]
  MoveL 462 to (-389.2, 700, 50) mm, rotated rx 180 ry 0 rz 90 deg; joints [-10.096, -73.569, 115.208, 33.113, 11.65, -40.448]
  MoveL 463 to (-389.2, 750, 50) mm, rotated rx 180 ry 0 rz 90 deg; joints [-10.431, -75.578, 117.927, 35.898, 11.205, -43.518]
  MoveL 464 to (-389.2, 750, -0.5) mm, rotated rx 180 ry 0 rz 90 deg; joints [-10.431, -73.497, 118.533, 45.684, 9.163, -53.458]
  MoveL 465 to (-389.2, 750, 50) mm, rotated rx 180 ry 0 rz 90 deg; joints [-10.431, -75.578, 117.927, 35.898, 11.205, -43.518]
  MoveL 466 to (-389.2, 800, 50) mm, rotated rx -180 ry 0 rz 90 deg; joints [-10.79, -77.616, 120.601, 38.707, 10.859, -46.627]
  MoveL 467 to (-389.2, 800, -0.5) mm, rotated rx -180 ry 0 rz 90 deg; joints [-10.79, -75.449, 121.224, 49.95, 8.853, -58.036]
  MoveL 468 to (-389.2, 800, 50) mm, rotated rx -180 ry 0 rz 90 deg; joints [-10.79, -77.616, 120.601, 38.707, 10.859, -46.627]
  MoveL 469 to (-389.2, 850, 50) mm, rotated rx 180 ry 0 rz 90 deg; joints [-11.174, -79.691, 123.231, 41.457, 10.615, -49.694]
  MoveL 470 to (-389.2, 850, -0.5) mm, rotated rx -180 ry 0 rz 90 deg; joints [-11.174, -77.432, 123.874, 54.15, 8.653, -62.565]
  MoveL 471 to (-389.2, 850, 50) mm, rotated rx 180 ry 0 rz 90 deg; joints [-11.174, -79.691, 123.231, 41.457, 10.615, -49.694]
  MoveL 472 to (-389.2, 900, 50) mm, rotated rx 180 ry 0 rz 90 deg; joints [-11.585, -81.811, 125.819, 44.05, 10.473, -52.621]
  MoveL 473 to (-389.2, 900, -0.5) mm, rotated rx -180 ry 0 rz 90 deg; joints [-11.585, -79.454, 126.484, 58.115, 8.56, -66.879]
  MoveL 474 to (-389.2, 900, 50) mm, rotated rx 180 ry 0 rz 90 deg; joints [-11.585, -81.811, 125.819, 44.05, 10.473, -52.621]
  MoveL 475 to (-389.2, 950, 50) mm, rotated rx 180 ry 0 rz 90 deg; joints [-12.028, -83.987, 128.366, 46.384, 10.437, -55.308]
  MoveL 476 to (-389.2, 950, -0.5) mm, rotated rx -180 ry 0 rz 90 deg; joints [-12.028, -81.525, 129.056, 61.673, 8.568, -70.806]
  MoveL 477 to (-389.2, 950, 50) mm, rotated rx 180 ry 0 rz 90 deg; joints [-12.028, -83.987, 128.366, 46.384, 10.437, -55.308]
  MoveL 478 to (-389.2, 1000, 50) mm, rotated rx -180 ry 0 rz 90 deg; joints [-12.506, -86.228, 130.873, 48.355, 10.507, -57.653]
  MoveL 479 to (-389.2, 1000, -0.5) mm, rotated rx -180 ry 0 rz 90 deg; joints [-12.506, -83.653, 131.591, 64.669, 8.671, -74.193]
  MoveL 480 to (-389.2, 1000, 50) mm, rotated rx -180 ry 0 rz 90 deg; joints [-12.506, -86.228, 130.873, 48.355, 10.507, -57.653]
  MoveL 481 to (-389.2, 1050, 50) mm, rotated rx 180 ry 0 rz 90 deg; joints [-13.022, -88.548, 133.341, 49.871, 10.688, -59.565]
  MoveL 482 to (-389.2, 1050, -0.5) mm, rotated rx 180 ry 0 rz 90 deg; joints [-13.022, -85.852, 134.09, 66.975, 8.863, -76.915]
  MoveL 483 to (-389.2, 1050, 50) mm, rotated rx 180 ry 0 rz 90 deg; joints [-13.022, -88.548, 133.341, 49.871, 10.688, -59.565]
  MoveL 484 to (-389.2, 1100, 50) mm, rotated rx 180 ry 0 rz 90 deg; joints [-13.581, -90.962, 135.769, 50.858, 10.984, -60.972]
  MoveL 485 to (-389.2, 1100, -0.5) mm, rotated rx -180 ry 0 rz 90 deg; joints [-13.581, -88.136, 136.553, 68.496, 9.139, -78.878]
  MoveL 486 to (-389.2, 1100, 50) mm, rotated rx 180 ry 0 rz 90 deg; joints [-13.581, -90.962, 135.769, 50.858, 10.984, -60.972]
  MoveL 487 to (-389.2, 1150, 50) mm, rotated rx 180 ry 0 rz 90 deg; joints [-14.19, -93.486, 138.156, 51.266, 11.407, -61.824]
  MoveL 488 to (-389.2, 1150, -0.5) mm, rotated rx 180 ry 0 rz 90 deg; joints [-14.19, -90.521, 138.98, 69.168, 9.501, -80.021]
  MoveL 489 to (-389.2, 1150, 50) mm, rotated rx 180 ry 0 rz 90 deg; joints [-14.19, -93.486, 138.156, 51.266, 11.407, -61.824]
  MoveL 490 to (-389.2, 1200, 50) mm, rotated rx -180 ry 0 rz 90 deg; joints [-14.855, -96.142, 140.502, 51.07, 11.97, -62.1]
  MoveL 491 to (-389.2, 1200, -0.5) mm, rotated rx -180 ry 0 rz 90 deg; joints [-14.855, -93.027, 141.37, 68.956, 9.955, -80.311]
  MoveL 492 to (-389.2, 1200, 50) mm, rotated rx -180 ry 0 rz 90 deg; joints [-14.855, -96.142, 140.502, 51.07, 11.97, -62.1]
  MoveL 493 to (-33.64, 230, 50) mm, rotated rx -180 ry 0 rz 90 deg; joints [-17.464, -51.672, 81.198, 26.405, 25.13, -37.944]
  MoveL 494 to (-33.64, 230, -0.5) mm, rotated rx 180 ry 0 rz 90 deg; joints [-17.464, -50.314, 81.725, 28.325, 23.456, -40.05]
  MoveL 495 to (-33.64, 230, 50) mm, rotated rx -180 ry 0 rz 90 deg; joints [-17.464, -51.672, 81.198, 26.405, 25.13, -37.944]
  MoveL 496 to (-63.64, 230, 50) mm, rotated rx -180 ry 0 rz 90 deg; joints [-16.675, -52.048, 81.835, 25.714, 24.595, -36.752]
  MoveL 497 to (-63.64, 230, -0.5) mm, rotated rx 180 ry 0 rz 90 deg; joints [-16.675, -50.681, 82.361, 27.646, 22.903, -38.862]
  MoveL 498 to (-63.64, 230, 50) mm, rotated rx -180 ry 0 rz 90 deg; joints [-16.675, -52.048, 81.835, 25.714, 24.595, -36.752]
  MoveL 499 to (-109.34, 230, 50) mm, rotated rx 180 ry 0 rz 90 deg; joints [-15.461, -52.585, 82.743, 24.552, 23.812, -34.813]
  MoveL 500 to (-109.34, 230, -0.5) mm, rotated rx -180 ry 0 rz 90 deg; joints [-15.461, -51.207, 83.269, 26.489, 22.094, -36.916]
  MoveL 501 to (-109.34, 230, 50) mm, rotated rx 180 ry 0 rz 90 deg; joints [-15.461, -52.585, 82.743, 24.552, 23.812, -34.813]
  MoveL 502 to (-139.34, 230, 50) mm, rotated rx 180 ry 0 rz 90 deg; joints [-14.655, -52.915, 83.299, 23.715, 23.321, -33.457]
  MoveL 503 to (-139.34, 230, -0.5) mm, rotated rx 180 ry 0 rz 90 deg; joints [-14.655, -51.53, 83.824, 25.646, 21.585, -35.546]
  MoveL 504 to (-139.34, 230, 50) mm, rotated rx 180 ry 0 rz 90 deg; joints [-14.655, -52.915, 83.299, 23.715, 23.321, -33.457]
  MoveL 505 to (-185.04, 230, 50) mm, rotated rx 180 ry 0 rz 90 deg; joints [-13.418, -53.382, 84.084, 22.322, 22.612, -31.261]
  MoveL 506 to (-185.04, 230, -0.5) mm, rotated rx 180 ry 0 rz 90 deg; joints [-13.418, -51.986, 84.609, 24.227, 20.847, -33.311]
  MoveL 507 to (-185.04, 230, 50) mm, rotated rx 180 ry 0 rz 90 deg; joints [-13.418, -53.382, 84.084, 22.322, 22.612, -31.261]
  MoveL 508 to (-215.04, 230, 50) mm, rotated rx 180 ry 0 rz 90 deg; joints [-12.598, -53.666, 84.56, 21.329, 22.172, -29.733]
  MoveL 509 to (-215.04, 230, -0.5) mm, rotated rx 180 ry 0 rz 90 deg; joints [-12.598, -52.263, 85.084, 23.204, 20.388, -31.744]
  MoveL 510 to (-215.04, 230, 50) mm, rotated rx 180 ry 0 rz 90 deg; joints [-12.598, -53.666, 84.56, 21.329, 22.172, -29.733]
  MoveL 511 to (-260.74, 230, 50) mm, rotated rx -180 ry 0 rz 90 deg; joints [-11.34, -54.062, 85.224, 19.693, 21.543, -27.271]
  MoveL 512 to (-260.74, 230, -0.5) mm, rotated rx -180 ry 0 rz 90 deg; joints [-11.34, -52.651, 85.748, 21.501, 19.731, -29.203]
  MoveL 513 to (-260.74, 230, 50) mm, rotated rx -180 ry 0 rz 90 deg; joints [-11.34, -54.062, 85.224, 19.693, 21.543, -27.271]
  MoveL 514 to (-290.74, 230, 50) mm, rotated rx 180 ry 0 rz 90 deg; joints [-10.507, -54.3, 85.62, 18.537, 21.16, -25.567]
  MoveL 515 to (-290.74, 230, -0.5) mm, rotated rx 180 ry 0 rz 90 deg; joints [-10.507, -52.883, 86.144, 20.287, 19.329, -27.431]
  MoveL 516 to (-290.74, 230, 50) mm, rotated rx 180 ry 0 rz 90 deg; joints [-10.507, -54.3, 85.62, 18.537, 21.16, -25.567]
  MoveL 517 to (-336.44, 230, 50) mm, rotated rx 180 ry 0 rz 90 deg; joints [-9.231, -54.626, 86.163, 16.655, 20.624, -22.84]
  MoveL 518 to (-336.44, 230, -0.5) mm, rotated rx 180 ry 0 rz 90 deg; joints [-9.231, -53.201, 86.687, 18.289, 18.765, -24.575]
  MoveL 519 to (-336.44, 230, 50) mm, rotated rx 180 ry 0 rz 90 deg; joints [-9.231, -54.626, 86.163, 16.655, 20.624, -22.84]
  MoveL 520 to (-366.44, 230, 50) mm, rotated rx 180 ry 0 rz 90 deg; joints [-8.388, -54.817, 86.481, 15.34, 20.304, -20.965]
  MoveL 521 to (-366.44, 230, -0.5) mm, rotated rx 180 ry 0 rz 90 deg; joints [-8.388, -53.388, 87.005, 16.882, 18.428, -22.599]
  MoveL 522 to (-366.44, 230, 50) mm, rotated rx 180 ry 0 rz 90 deg; joints [-8.388, -54.817, 86.481, 15.34, 20.304, -20.965]
  MoveL 523 to (-33.64, 420, 50) mm, rotated rx -180 ry 0 rz 90 deg; joints [-19.177, -59.135, 93.55, 34.115, 21.629, -47.325]
  MoveL 524 to (-33.64, 420, -0.5) mm, rotated rx -180 ry 0 rz 90 deg; joints [-19.177, -57.599, 94.076, 37.285, 19.954, -50.715]
  MoveL 525 to (-33.64, 420, 50) mm, rotated rx -180 ry 0 rz 90 deg; joints [-19.177, -59.135, 93.55, 34.115, 21.629, -47.325]
  MoveL 526 to (-63.64, 420, 50) mm, rotated rx 180 ry 0 rz 90 deg; joints [-18.322, -59.523, 94.174, 33.435, 21.041, -46.074]
  MoveL 527 to (-63.64, 420, -0.5) mm, rotated rx -180 ry 0 rz 90 deg; joints [-18.322, -57.977, 94.701, 36.674, 19.343, -49.524]
  MoveL 528 to (-63.64, 420, 50) mm, rotated rx 180 ry 0 rz 90 deg; joints [-18.322, -59.523, 94.174, 33.435, 21.041, -46.074]
  MoveL 529 to (-109.34, 420, 50) mm, rotated rx -180 ry 0 rz 90 deg; joints [-17.002, -60.08, 95.066, 32.251, 20.172, -44.004]
  MoveL 530 to (-109.34, 420, -0.5) mm, rotated rx -180 ry 0 rz 90 deg; joints [-17.002, -58.519, 95.594, 35.579, 18.437, -47.53]
  MoveL 531 to (-109.34, 420, 50) mm, rotated rx -180 ry 0 rz 90 deg; joints [-17.002, -60.08, 95.066, 32.251, 20.172, -44.004]
  MoveL 532 to (-139.34, 420, 50) mm, rotated rx -180 ry 0 rz 90 deg; joints [-16.125, -60.423, 95.613, 31.367, 19.62, -42.528]
  MoveL 533 to (-139.34, 420, -0.5) mm, rotated rx 180 ry 0 rz 90 deg; joints [-16.125, -58.852, 96.142, 34.743, 17.86, -46.092]
  MoveL 534 to (-139.34, 420, 50) mm, rotated rx -180 ry 0 rz 90 deg; joints [-16.125, -60.423, 95.613, 31.367, 19.62, -42.528]
  MoveL 535 to (-185.04, 420, 50) mm, rotated rx 180 ry 0 rz 90 deg; joints [-14.774, -60.91, 96.388, 29.847, 18.812, -40.091]
  MoveL 536 to (-185.04, 420, -0.5) mm, rotated rx -180 ry 0 rz 90 deg; joints [-14.774, -59.326, 96.918, 33.27, 17.01, -43.688]
  MoveL 537 to (-185.04, 420, 50) mm, rotated rx 180 ry 0 rz 90 deg; joints [-14.774, -60.91, 96.388, 29.847, 18.812, -40.091]
  MoveL 538 to (-215.04, 420, 50) mm, rotated rx 180 ry 0 rz 90 deg; joints [-13.878, -61.207, 96.858, 28.727, 18.304, -38.36]
  MoveL 539 to (-215.04, 420, -0.5) mm, rotated rx 180 ry 0 rz 90 deg; joints [-13.878, -59.615, 97.388, 32.162, 16.473, -41.959]
  MoveL 540 to (-215.04, 420, 50) mm, rotated rx 180 ry 0 rz 90 deg; joints [-13.878, -61.207, 96.858, 28.727, 18.304, -38.36]
  MoveL 541 to (-260.74, 420, 50) mm, rotated rx -180 ry 0 rz 90 deg; joints [-12.5, -61.623, 97.515, 26.823, 17.569, -35.512]
  MoveL 542 to (-260.74, 420, -0.5) mm, rotated rx -180 ry 0 rz 90 deg; joints [-12.5, -60.019, 98.047, 30.238, 15.693, -39.075]
  MoveL 543 to (-260.74, 420, 50) mm, rotated rx -180 ry 0 rz 90 deg; joints [-12.5, -61.623, 97.515, 26.823, 17.569, -35.512]
  MoveL 544 to (-290.74, 420, 50) mm, rotated rx -180 ry 0 rz 90 deg; joints [-11.587, -61.873, 97.908, 25.437, 17.115, -33.499]
  MoveL 545 to (-290.74, 420, -0.5) mm, rotated rx 180 ry 0 rz 90 deg; joints [-11.587, -60.262, 98.44, 28.809, 15.207, -37.009]
  MoveL 546 to (-290.74, 420, 50) mm, rotated rx -180 ry 0 rz 90 deg; joints [-11.587, -61.873, 97.908, 25.437, 17.115, -33.499]
  MoveL 547 to (-336.44, 420, 50) mm, rotated rx 180 ry 0 rz 90 deg; joints [-10.185, -62.216, 98.448, 23.11, 16.47, -30.205]
  MoveL 548 to (-336.44, 420, -0.5) mm, rotated rx 180 ry 0 rz 90 deg; joints [-10.185, -60.596, 98.981, 26.362, 14.514, -33.578]
  MoveL 549 to (-336.44, 420, 50) mm, rotated rx 180 ry 0 rz 90 deg; joints [-10.185, -62.216, 98.448, 23.11, 16.47, -30.205]
  MoveL 550 to (-366.44, 420, 50) mm, rotated rx -180 ry 0 rz 90 deg; joints [-9.258, -62.418, 98.764, 21.439, 16.081, -27.892]
  MoveL 551 to (-366.44, 420, -0.5) mm, rotated rx 180 ry 0 rz 90 deg; joints [-9.258, -60.792, 99.298, 24.57, 14.093, -31.134]
  MoveL 552 to (-366.44, 420, 50) mm, rotated rx -180 ry 0 rz 90 deg; joints [-9.258, -62.418, 98.764, 21.439, 16.081, -27.892]
  MoveL 553 to (-33.64, 730, 50) mm, rotated rx -180 ry 0 rz 90 deg; joints [-22.788, -70.66, 111.128, 48.63, 18.953, -65.123]
  MoveL 554 to (-33.64, 730, -0.5) mm, rotated rx 180 ry 0 rz 90 deg; joints [-22.788, -68.767, 111.698, 54.505, 17.421, -71.305]
  MoveL 555 to (-33.64, 730, 50) mm, rotated rx -180 ry 0 rz 90 deg; joints [-22.788, -70.66, 111.128, 48.63, 18.953, -65.123]
  MoveL 556 to (-63.64, 730, 50) mm, rotated rx -180 ry 0 rz 90 deg; joints [-21.801, -71.115, 111.777, 48.225, 18.264, -64.018]
  MoveL 557 to (-63.64, 730, -0.5) mm, rotated rx -180 ry 0 rz 90 deg; joints [-21.801, -69.206, 112.35, 54.377, 16.71, -70.467]
  MoveL 558 to (-63.64, 730, 50) mm, rotated rx -180 ry 0 rz 90 deg; joints [-21.801, -71.115, 111.777, 48.225, 18.264, -64.018]
  MoveL 559 to (-109.34, 730, 50) mm, rotated rx -180 ry 0 rz 90 deg; joints [-20.271, -71.773, 112.708, 47.427, 17.222, -62.131]
  MoveL 560 to (-109.34, 730, -0.5) mm, rotated rx 180 ry 0 rz 90 deg; joints [-20.271, -69.84, 113.285, 54.023, 15.63, -69.006]
  MoveL 561 to (-109.34, 730, 50) mm, rotated rx -180 ry 0 rz 90 deg; joints [-20.271, -71.773, 112.708, 47.427, 17.222, -62.131]
  MoveL 562 to (-139.34, 730, 50) mm, rotated rx -180 ry 0 rz 90 deg; joints [-19.25, -72.181, 113.281, 46.768, 16.545, -60.741]
  MoveL 563 to (-139.34, 730, -0.5) mm, rotated rx 180 ry 0 rz 90 deg; joints [-19.25, -70.233, 113.861, 53.669, 14.924, -67.91]
  MoveL 564 to (-139.34, 730, 50) mm, rotated rx -180 ry 0 rz 90 deg; joints [-19.25, -72.181, 113.281, 46.768, 16.545, -60.741]
  MoveL 565 to (-185.04, 730, 50) mm, rotated rx -180 ry 0 rz 90 deg; joints [-17.67, -72.764, 114.095, 45.523, 15.528, -58.363]
  MoveL 566 to (-185.04, 730, -0.5) mm, rotated rx -180 ry 0 rz 90 deg; joints [-17.67, -70.794, 114.679, 52.905, 13.856, -65.993]
  MoveL 567 to (-185.04, 730, 50) mm, rotated rx -180 ry 0 rz 90 deg; joints [-17.67, -72.764, 114.095, 45.523, 15.528, -58.363]
  MoveL 568 to (-215.04, 730, 50) mm, rotated rx 180 ry 0 rz 90 deg; joints [-16.617, -73.121, 114.59, 44.524, 14.872, -56.606]
  MoveL 569 to (-215.04, 730, -0.5) mm, rotated rx 180 ry 0 rz 90 deg; joints [-16.617, -71.138, 115.177, 52.229, 13.16, -64.546]
  MoveL 570 to (-215.04, 730, 50) mm, rotated rx 180 ry 0 rz 90 deg; joints [-16.617, -73.121, 114.59, 44.524, 14.872, -56.606]
  MoveL 571 to (-260.74, 730, 50) mm, rotated rx 180 ry 0 rz 90 deg; joints [-14.992, -73.626, 115.285, 42.68, 13.895, -53.589]
  MoveL 572 to (-260.74, 730, -0.5) mm, rotated rx 180 ry 0 rz 90 deg; joints [-14.992, -71.622, 115.876, 50.872, 12.114, -61.996]
  MoveL 573 to (-260.74, 730, 50) mm, rotated rx 180 ry 0 rz 90 deg; joints [-14.992, -73.626, 115.285, 42.68, 13.895, -53.589]
  MoveL 574 to (-290.74, 730, 50) mm, rotated rx 180 ry 0 rz 90 deg; joints [-13.91, -73.93, 115.702, 41.226, 13.272, -51.354]
  MoveL 575 to (-290.74, 730, -0.5) mm, rotated rx 180 ry 0 rz 90 deg; joints [-13.91, -71.914, 116.294, 49.725, 11.438, -60.052]
  MoveL 576 to (-290.74, 730, 50) mm, rotated rx 180 ry 0 rz 90 deg; joints [-13.91, -73.93, 115.702, 41.226, 13.272, -51.354]
  MoveL 577 to (-336.44, 730, 50) mm, rotated rx 180 ry 0 rz 90 deg; joints [-12.244, -74.351, 116.275, 38.582, 12.358, -47.502]
  MoveL 578 to (-336.44, 730, -0.5) mm, rotated rx 180 ry 0 rz 90 deg; joints [-12.244, -72.319, 116.871, 47.491, 10.431, -56.589]
  MoveL 579 to (-336.44, 730, 50) mm, rotated rx 180 ry 0 rz 90 deg; joints [-12.244, -74.351, 116.275, 38.582, 12.358, -47.502]
  MoveL 580 to (-366.44, 730, 50) mm, rotated rx 180 ry 0 rz 90 deg; joints [-11.139, -74.599, 116.612, 36.526, 11.787, -44.643]
  MoveL 581 to (-366.44, 730, -0.5) mm, rotated rx 180 ry 0 rz 90 deg; joints [-11.139, -72.557, 117.209, 45.64, 9.79, -53.92]
  MoveL 582 to (-366.44, 730, 50) mm, rotated rx 180 ry 0 rz 90 deg; joints [-11.139, -74.599, 116.612, 36.526, 11.787, -44.643]
  MoveL 583 to (-33.64, 1020, 50) mm, rotated rx 180 ry 0 rz 90 deg; joints [-27.545, -81.546, 125.501, 59.392, 19.763, -79.91]
  MoveL 584 to (-33.64, 1020, -0.5) mm, rotated rx -180 ry 0 rz 90 deg; joints [-27.545, -79.202, 126.164, 67.162, 18.408, -88.129]
  MoveL 585 to (-33.64, 1020, 50) mm, rotated rx 180 ry 0 rz 90 deg; joints [-27.545, -81.546, 125.501, 59.392, 19.763, -79.91]
  MoveL 586 to (-63.64, 1020, 50) mm, rotated rx -180 ry 0 rz 90 deg; joints [-26.408, -82.143, 126.214, 59.282, 19.001, -78.956]
  MoveL 587 to (-63.64, 1020, -0.5) mm, rotated rx 180 ry 0 rz 90 deg; joints [-26.408, -79.77, 126.883, 67.505, 17.635, -87.616]
  MoveL 588 to (-63.64, 1020, 50) mm, rotated rx -180 ry 0 rz 90 deg; joints [-26.408, -82.143, 126.214, 59.282, 19.001, -78.956]
  MoveL 589 to (-109.34, 1020, 50) mm, rotated rx 180 ry 0 rz 90 deg; joints [-24.633, -83.014, 127.241, 58.955, 17.827, -77.308]
  MoveL 590 to (-109.34, 1020, -0.5) mm, rotated rx 180 ry 0 rz 90 deg; joints [-24.633, -80.6, 127.92, 67.942, 16.44, -86.71]
  MoveL 591 to (-109.34, 1020, 50) mm, rotated rx 180 ry 0 rz 90 deg; joints [-24.633, -83.014, 127.241, 58.955, 17.827, -77.308]
  MoveL 592 to (-139.34, 1020, 50) mm, rotated rx 180 ry 0 rz 90 deg; joints [-23.439, -83.56, 127.875, 58.619, 17.051, -76.083]
  MoveL 593 to (-139.34, 1020, -0.5) mm, rotated rx 180 ry 0 rz 90 deg; joints [-23.439, -81.119, 128.561, 68.161, 15.645, -86.024]
  MoveL 594 to (-139.34, 1020, 50) mm, rotated rx 180 ry 0 rz 90 deg; joints [-23.439, -83.56, 127.875, 58.619, 17.051, -76.083]
  MoveL 595 to (-185.04, 1020, 50) mm, rotated rx -180 ry 0 rz 90 deg; joints [-21.578, -84.349, 128.78, 57.882, 15.859, -73.958]
  MoveL 596 to (-185.04, 1020, -0.5) mm, rotated rx 180 ry 0 rz 90 deg; joints [-21.578, -81.87, 129.474, 68.366, 14.417, -84.815]
  MoveL 597 to (-185.04, 1020, 50) mm, rotated rx -180 ry 0 rz 90 deg; joints [-21.578, -84.349, 128.78, 57.882, 15.859, -73.958]
  MoveL 598 to (-215.04, 1020, 50) mm, rotated rx -180 ry 0 rz 90 deg; joints [-20.33, -84.838, 129.332, 57.224, 15.073, -72.368]
  MoveL 599 to (-215.04, 1020, -0.5) mm, rotated rx 180 ry 0 rz 90 deg; joints [-20.33, -82.334, 130.033, 68.398, 13.601, -83.898]
  MoveL 600 to (-215.04, 1020, 50) mm, rotated rx -180 ry 0 rz 90 deg; joints [-20.33, -84.838, 129.332, 57.224, 15.073, -72.368]
  MoveL 601 to (-260.74, 1020, 50) mm, rotated rx -180 ry 0 rz 90 deg; joints [-18.39, -85.534, 130.109, 55.894, 13.873, -69.589]
  MoveL 602 to (-260.74, 1020, -0.5) mm, rotated rx 180 ry 0 rz 90 deg; joints [-18.39, -82.994, 130.818, 68.247, 12.343, -82.269]
  MoveL 603 to (-260.74, 1020, 50) mm, rotated rx -180 ry 0 rz 90 deg; joints [-18.39, -85.534, 130.109, 55.894, 13.873, -69.589]
  MoveL 604 to (-290.74, 1020, 50) mm, rotated rx 180 ry 0 rz 90 deg; joints [-17.091, -85.957, 130.576, 54.762, 13.088, -67.487]
  MoveL 605 to (-290.74, 1020, -0.5) mm, rotated rx 180 ry 0 rz 90 deg; joints [-17.091, -83.396, 131.291, 67.983, 11.508, -81.015]
  MoveL 606 to (-290.74, 1020, 50) mm, rotated rx 180 ry 0 rz 90 deg; joints [-17.091, -85.957, 130.576, 54.762, 13.088, -67.487]
  MoveL 607 to (-336.44, 1020, 50) mm, rotated rx -180 ry 0 rz 90 deg; joints [-15.079, -86.548, 131.222, 52.542, 11.902, -63.765]
  MoveL 608 to (-336.44, 1020, -0.5) mm, rotated rx 180 ry 0 rz 90 deg; joints [-15.079, -83.957, 131.944, 67.245, 10.226, -78.742]
  MoveL 609 to (-336.44, 1020, 50) mm, rotated rx -180 ry 0 rz 90 deg; joints [-15.079, -86.548, 131.222, 52.542, 11.902, -63.765]
  MoveL 610 to (-366.44, 1020, 50) mm, rotated rx -180 ry 0 rz 90 deg; joints [-13.736, -86.9, 131.601, 50.685, 11.136, -60.906]
  MoveL 611 to (-366.44, 1020, -0.5) mm, rotated rx -180 ry 0 rz 90 deg; joints [-13.736, -84.29, 132.328, 66.47, 9.38, -76.943]
  MoveL 612 to (-366.44, 1020, 50) mm, rotated rx -180 ry 0 rz 90 deg; joints [-13.736, -86.9, 131.601, 50.685, 11.136, -60.906]
  MoveL 613 to (-450, 50, 50) mm, rotated rx 180 ry 0 rz 90 deg; joints [-5.525, -47.551, 74.124, 8.31, 24.787, -11.853]
  MoveL 614 to (-450, 50, -0.5) mm, rotated rx -180 ry 0 rz 90 deg; joints [-5.525, -46.278, 74.662, 8.923, 22.996, -12.523]
  MoveL 615 to (-450, 50, 50) mm, rotated rx 180 ry 0 rz 90 deg; joints [-5.525, -47.551, 74.124, 8.31, 24.787, -11.853]
  MoveL 616 to (-450, 100, 50) mm, rotated rx -180 ry 0 rz 90 deg; joints [-5.655, -49.761, 77.937, 9.049, 23.219, -12.727]
  MoveL 617 to (-450, 100, -0.5) mm, rotated rx 180 ry 0 rz 90 deg; joints [-5.655, -48.443, 78.469, 9.787, 21.395, -13.524]
  MoveL 618 to (-450, 100, 50) mm, rotated rx -180 ry 0 rz 90 deg; joints [-5.655, -49.761, 77.937, 9.049, 23.219, -12.727]
  MoveL 619 to (-450, 150, 50) mm, rotated rx 180 ry 0 rz 90 deg; joints [-5.79, -51.91, 81.602, 9.868, 21.744, -13.684]
  MoveL 620 to (-450, 150, -0.5) mm, rotated rx 180 ry 0 rz 90 deg; joints [-5.79, -50.547, 82.129, 10.758, 19.884, -14.637]
  MoveL 621 to (-450, 150, 50) mm, rotated rx 180 ry 0 rz 90 deg; joints [-5.79, -51.91, 81.602, 9.868, 21.744, -13.684]
  MoveL 622 to (-450, 200, 50) mm, rotated rx 180 ry 0 rz 90 deg; joints [-5.932, -54.011, 85.137, 10.778, 20.354, -14.736]
  MoveL 623 to (-450, 200, -0.5) mm, rotated rx 180 ry 0 rz 90 deg; joints [-5.932, -52.6, 85.661, 11.856, 18.457, -15.879]
  MoveL 624 to (-450, 200, 50) mm, rotated rx 180 ry 0 rz 90 deg; joints [-5.932, -54.011, 85.137, 10.778, 20.354, -14.736]
  MoveL 625 to (-450, 250, 50) mm, rotated rx -180 ry 0 rz 90 deg; joints [-6.082, -56.071, 88.557, 11.79, 19.045, -15.895]
  MoveL 626 to (-450, 250, -0.5) mm, rotated rx -180 ry 0 rz 90 deg; joints [-6.082, -54.612, 89.081, 13.099, 17.109, -17.272]
  MoveL 627 to (-450, 250, 50) mm, rotated rx -180 ry 0 rz 90 deg; joints [-6.082, -56.071, 88.557, 11.79, 19.045, -15.895]
  MoveL 628 to (-450, 300, 50) mm, rotated rx 180 ry 0 rz 90 deg; joints [-6.239, -58.099, 91.875, 12.918, 17.813, -17.174]
  MoveL 629 to (-450, 300, -0.5) mm, rotated rx 180 ry 0 rz 90 deg; joints [-6.239, -56.59, 92.4, 14.513, 15.837, -18.841]
  MoveL 630 to (-450, 300, 50) mm, rotated rx 180 ry 0 rz 90 deg; joints [-6.239, -58.099, 91.875, 12.918, 17.813, -17.174]
  MoveL 631 to (-450, 350, 50) mm, rotated rx 180 ry 0 rz 90 deg; joints [-6.404, -60.102, 95.102, 14.176, 16.656, -18.589]
  MoveL 632 to (-450, 350, -0.5) mm, rotated rx 180 ry 0 rz 90 deg; joints [-6.404, -58.54, 95.63, 16.127, 14.639, -20.614]
  MoveL 633 to (-450, 350, 50) mm, rotated rx 180 ry 0 rz 90 deg; joints [-6.404, -60.102, 95.102, 14.176, 16.656, -18.589]
  MoveL 634 to (-450, 400, 50) mm, rotated rx 180 ry 0 rz 90 deg; joints [-6.579, -62.088, 98.246, 15.579, 15.572, -20.155]
  MoveL 635 to (-450, 400, -0.5) mm, rotated rx 180 ry 0 rz 90 deg; joints [-6.579, -60.471, 98.779, 17.971, 13.514, -22.626]
  MoveL 636 to (-450, 400, 50) mm, rotated rx 180 ry 0 rz 90 deg; joints [-6.579, -62.088, 98.246, 15.579, 15.572, -20.155]
  MoveL 637 to (-450, 450, 50) mm, rotated rx -180 ry 0 rz 90 deg; joints [-6.763, -64.061, 101.316, 17.142, 14.562, -21.888]
  MoveL 638 to (-450, 450, -0.5) mm, rotated rx 180 ry 0 rz 90 deg; joints [-6.763, -62.386, 101.854, 20.082, 12.464, -24.911]
  MoveL 639 to (-450, 450, 50) mm, rotated rx -180 ry 0 rz 90 deg; joints [-6.763, -64.061, 101.316, 17.142, 14.562, -21.888]
  MoveL 640 to (-450, 500, 50) mm, rotated rx 180 ry 0 rz 90 deg; joints [-6.957, -66.028, 104.317, 18.879, 13.626, -23.801]
  MoveL 641 to (-450, 500, -0.5) mm, rotated rx 180 ry 0 rz 90 deg; joints [-6.957, -64.293, 104.863, 22.498, 11.491, -27.508]
  MoveL 642 to (-450, 500, 50) mm, rotated rx 180 ry 0 rz 90 deg; joints [-6.957, -66.028, 104.317, 18.879, 13.626, -23.801]
  MoveL 643 to (-450, 550, 50) mm, rotated rx 180 ry 0 rz 90 deg; joints [-7.163, -67.995, 107.255, 20.799, 12.767, -25.906]
  MoveL 644 to (-450, 550, -0.5) mm, rotated rx -180 ry 0 rz 90 deg; joints [-7.163, -66.196, 107.81, 25.256, 10.598, -30.456]
  MoveL 645 to (-450, 550, 50) mm, rotated rx 180 ry 0 rz 90 deg; joints [-7.163, -67.995, 107.255, 20.799, 12.767, -25.906]
  MoveL 646 to (-450, 600, 50) mm, rotated rx 180 ry 0 rz 90 deg; joints [-7.382, -69.968, 110.135, 22.91, 11.988, -28.21]
  MoveL 647 to (-450, 600, -0.5) mm, rotated rx 180 ry 0 rz 90 deg; joints [-7.382, -68.101, 110.701, 28.388, 9.791, -33.788]
  MoveL 648 to (-450, 600, 50) mm, rotated rx 180 ry 0 rz 90 deg; joints [-7.382, -69.968, 110.135, 22.91, 11.988, -28.21]
  MoveL 649 to (-450, 650, 50) mm, rotated rx -180 ry 0 rz 90 deg; joints [-7.614, -71.952, 112.96, 25.206, 11.291, -30.708]
  MoveL 650 to (-450, 650, -0.5) mm, rotated rx 180 ry 0 rz 90 deg; joints [-7.614, -70.013, 113.539, 31.913, 9.075, -37.521]
  MoveL 651 to (-450, 650, 50) mm, rotated rx -180 ry 0 rz 90 deg; joints [-7.614, -71.952, 112.96, 25.206, 11.291, -30.708]
  MoveL 652 to (-450, 700, 50) mm, rotated rx -180 ry 0 rz 90 deg; joints [-7.861, -73.955, 115.736, 27.672, 10.681, -33.386]
  MoveL 653 to (-450, 700, -0.5) mm, rotated rx 180 ry 0 rz 90 deg; joints [-7.861, -71.938, 116.329, 35.824, 8.457, -41.652]
  MoveL 654 to (-450, 700, 50) mm, rotated rx -180 ry 0 rz 90 deg; joints [-7.861, -73.955, 115.736, 27.672, 10.681, -33.386]
  MoveL 655 to (-450, 750, 50) mm, rotated rx -180 ry 0 rz 90 deg; joints [-8.125, -75.982, 118.464, 30.271, 10.163, -36.21]
  MoveL 656 to (-450, 750, -0.5) mm, rotated rx -180 ry 0 rz 90 deg; joints [-8.125, -73.884, 119.073, 40.074, 7.941, -46.133]
  MoveL 657 to (-450, 750, 50) mm, rotated rx -180 ry 0 rz 90 deg; joints [-8.125, -75.982, 118.464, 30.271, 10.163, -36.21]
  MoveL 658 to (-450, 800, 50) mm, rotated rx 180 ry 0 rz 90 deg; joints [-8.407, -78.041, 121.148, 32.949, 9.739, -39.122]
  MoveL 659 to (-450, 800, -0.5) mm, rotated rx -180 ry 0 rz 90 deg; joints [-8.407, -75.856, 121.775, 44.564, 7.534, -50.867]
  MoveL 660 to (-450, 800, 50) mm, rotated rx 180 ry 0 rz 90 deg; joints [-8.407, -78.041, 121.148, 32.949, 9.739, -39.122]
  MoveL 661 to (-450, 850, 50) mm, rotated rx 180 ry 0 rz 90 deg; joints [-8.709, -80.141, 123.788, 35.624, 9.416, -42.045]
  MoveL 662 to (-450, 850, -0.5) mm, rotated rx -180 ry 0 rz 90 deg; joints [-8.709, -77.862, 124.436, 49.137, 7.238, -55.699]
  MoveL 663 to (-450, 850, 50) mm, rotated rx 180 ry 0 rz 90 deg; joints [-8.709, -80.141, 123.788, 35.624, 9.416, -42.045]
  MoveL 664 to (-450, 900, 50) mm, rotated rx 180 ry 0 rz 90 deg; joints [-9.033, -82.29, 126.388, 38.194, 9.195, -44.877]
  MoveL 665 to (-450, 900, -0.5) mm, rotated rx 180 ry 0 rz 90 deg; joints [-9.033, -79.91, 127.059, 53.585, 7.053, -60.42]
  MoveL 666 to (-450, 900, 50) mm, rotated rx 180 ry 0 rz 90 deg; joints [-9.033, -82.29, 126.388, 38.194, 9.195, -44.877]
  MoveL 667 to (-450, 950, 50) mm, rotated rx 180 ry 0 rz 90 deg; joints [-9.382, -84.498, 128.949, 40.539, 9.082, -47.499]
  MoveL 668 to (-450, 950, -0.5) mm, rotated rx 180 ry 0 rz 90 deg; joints [-9.382, -82.011, 129.645, 57.67, 6.974, -64.794]
  MoveL 669 to (-450, 950, 50) mm, rotated rx 180 ry 0 rz 90 deg; joints [-9.382, -84.498, 128.949, 40.539, 9.082, -47.499]
  MoveL 670 to (-450, 1000, 50) mm, rotated rx 180 ry 0 rz 90 deg; joints [-9.759, -86.778, 131.47, 42.533, 9.079, -49.787]
  MoveL 671 to (-450, 1000, -0.5) mm, rotated rx 180 ry 0 rz 90 deg; joints [-9.759, -84.175, 132.196, 61.155, 6.995, -68.587]
  MoveL 672 to (-450, 1000, 50) mm, rotated rx 180 ry 0 rz 90 deg; joints [-9.759, -86.778, 131.47, 42.533, 9.079, -49.787]
  MoveL 673 to (-450, 1050, 50) mm, rotated rx -180 ry 0 rz 90 deg; joints [-10.168, -89.144, 133.954, 44.059, 9.192, -51.624]
  MoveL 674 to (-450, 1050, -0.5) mm, rotated rx 180 ry 0 rz 90 deg; joints [-10.168, -86.417, 134.711, 63.836, 7.11, -71.595]
  MoveL 675 to (-450, 1050, 50) mm, rotated rx -180 ry 0 rz 90 deg; joints [-10.168, -89.144, 133.954, 44.059, 9.192, -51.624]
  MoveL 676 to (-450, 1100, 50) mm, rotated rx 180 ry 0 rz 90 deg; joints [-10.611, -91.612, 136.399, 45.018, 9.429, -52.911]
  MoveL 677 to (-450, 1100, -0.5) mm, rotated rx 180 ry 0 rz 90 deg; joints [-10.611, -88.751, 137.193, 65.554, 7.313, -73.661]
  MoveL 678 to (-450, 1100, 50) mm, rotated rx 180 ry 0 rz 90 deg; joints [-10.611, -91.612, 136.399, 45.018, 9.429, -52.911]
  MoveL 679 to (-450, 1150, 50) mm, rotated rx 180 ry 0 rz 90 deg; joints [-11.094, -94.201, 138.805, 45.34, 9.802, -53.584]
  MoveL 680 to (-450, 1150, -0.5) mm, rotated rx -180 ry 0 rz 90 deg; joints [-11.094, -91.196, 139.64, 66.205, 7.605, -74.683]
  MoveL 681 to (-450, 1150, 50) mm, rotated rx 180 ry 0 rz 90 deg; joints [-11.094, -94.201, 138.805, 45.34, 9.802, -53.584]
  MoveL 682 to (-450, 1200, 50) mm, rotated rx -180 ry 0 rz 90 deg; joints [-11.623, -96.935, 141.171, 44.999, 10.33, -53.613]
  MoveL 683 to (-450, 1200, -0.5) mm, rotated rx -180 ry 0 rz 90 deg; joints [-11.623, -93.776, 142.052, 65.736, 7.995, -74.608]
  MoveL 684 to (-450, 1200, 50) mm, rotated rx -180 ry 0 rz 90 deg; joints [-11.623, -96.935, 141.171, 44.999, 10.33, -53.613]
  MoveL 685 to (-450, 1250, 50) mm, rotated rx 180 ry 0 rz 90 deg; joints [-12.204, -99.842, 143.493, 44.01, 11.039, -53.016]
  MoveL 686 to (-450, 1250, -0.5) mm, rotated rx 180 ry 0 rz 90 deg; joints [-12.204, -96.518, 144.428, 64.144, 8.502, -73.436]
  MoveL 687 to (-450, 1250, 50) mm, rotated rx 180 ry 0 rz 90 deg; joints [-12.204, -99.842, 143.493, 44.01, 11.039, -53.016]
  MoveL 688 to (-450, 1300, 50) mm, rotated rx 180 ry 0 rz 90 deg; joints [-12.845, -102.955, 145.77, 42.43, 11.968, -51.853]
  MoveL 689 to (-450, 1300, -0.5) mm, rotated rx 180 ry 0 rz 90 deg; joints [-12.845, -99.459, 146.765, 61.487, 9.162, -71.227]
  MoveL 690 to (-450, 1300, 50) mm, rotated rx 180 ry 0 rz 90 deg; joints [-12.845, -102.955, 145.77, 42.43, 11.968, -51.853]
  MoveL 691 to (-450, 1350, 50) mm, rotated rx -180 ry 0 rz 90 deg; joints [-13.556, -106.315, 147.997, 40.359, 13.167, -50.22]
  MoveL 692 to (-450, 1350, -0.5) mm, rotated rx 180 ry 0 rz 90 deg; joints [-13.556, -102.64, 149.059, 57.89, 10.029, -68.105]
  MoveL 693 to (-450, 1350, 50) mm, rotated rx -180 ry 0 rz 90 deg; joints [-13.556, -106.315, 147.997, 40.359, 13.167, -50.22]
  MoveL 694 to (-450, 1400, 50) mm, rotated rx -180 ry 0 rz 90 deg; joints [-14.349, -109.974, 150.166, 37.922, 14.7, -48.245]
  MoveL 695 to (-450, 1400, -0.5) mm, rotated rx 180 ry 0 rz 90 deg; joints [-14.349, -106.119, 151.307, 53.552, 11.18, -64.27]
  MoveL 696 to (-450, 1400, 50) mm, rotated rx -180 ry 0 rz 90 deg; joints [-14.349, -109.974, 150.166, 37.922, 14.7, -48.245]
  MoveL 697 to (-450, 1450, 50) mm, rotated rx 180 ry 0 rz 90 deg; joints [-15.237, -113.991, 152.269, 35.264, 16.647, -46.068]
  MoveL 698 to (-450, 1450, -0.5) mm, rotated rx -180 ry 0 rz 90 deg; joints [-15.237, -109.964, 153.501, 48.736, 12.711, -59.982]
  MoveL 699 to (-450, 1450, 50) mm, rotated rx 180 ry 0 rz 90 deg; joints [-15.237, -113.991, 152.269, 35.264, 16.647, -46.068]
  MoveL 700 to (-578.4, 50, 50) mm, rotated rx 180 ry 0 rz 90 deg; joints [-2.153, -47.938, 74.794, 3.306, 24.199, -4.689]
  MoveL 701 to (-578.4, 50, -0.5) mm, rotated rx 180 ry 0 rz 90 deg; joints [-2.153, -46.657, 75.332, 3.559, 22.384, -4.964]
  MoveL 702 to (-578.4, 50, 50) mm, rotated rx 180 ry 0 rz 90 deg; joints [-2.153, -47.938, 74.794, 3.306, 24.199, -4.689]
  MoveL 703 to (-578.4, 100, 50) mm, rotated rx -180 ry 0 rz 90 deg; joints [-2.203, -50.145, 78.596, 3.608, 22.61, -5.044]
  MoveL 704 to (-578.4, 100, -0.5) mm, rotated rx 180 ry 0 rz 90 deg; joints [-2.203, -48.82, 79.126, 3.914, 20.758, -5.373]
  MoveL 705 to (-578.4, 100, 50) mm, rotated rx -180 ry 0 rz 90 deg; joints [-2.203, -50.145, 78.596, 3.608, 22.61, -5.044]
  MoveL 706 to (-578.4, 150, 50) mm, rotated rx 180 ry 0 rz 90 deg; joints [-2.256, -52.294, 82.252, 3.945, 21.11, -5.435]
  MoveL 707 to (-578.4, 150, -0.5) mm, rotated rx -180 ry 0 rz 90 deg; joints [-2.256, -50.922, 82.778, 4.317, 19.217, -5.831]
  MoveL 708 to (-578.4, 150, 50) mm, rotated rx 180 ry 0 rz 90 deg; joints [-2.256, -52.294, 82.252, 3.945, 21.11, -5.435]
  MoveL 709 to (-578.4, 200, 50) mm, rotated rx -180 ry 0 rz 90 deg; joints [-2.312, -54.396, 85.78, 4.322, 19.69, -5.867]
  MoveL 710 to (-578.4, 200, -0.5) mm, rotated rx -180 ry 0 rz 90 deg; joints [-2.312, -52.977, 86.304, 4.776, 17.753, -6.347]
  MoveL 711 to (-578.4, 200, 50) mm, rotated rx -180 ry 0 rz 90 deg; joints [-2.312, -54.396, 85.78, 4.322, 19.69, -5.867]
  MoveL 712 to (-578.4, 250, 50) mm, rotated rx -180 ry 0 rz 90 deg; joints [-2.371, -56.459, 89.196, 4.744, 18.345, -6.347]
  MoveL 713 to (-578.4, 250, -0.5) mm, rotated rx 180 ry 0 rz 90 deg; joints [-2.371, -54.991, 89.72, 5.303, 16.361, -6.932]
  MoveL 714 to (-578.4, 250, 50) mm, rotated rx -180 ry 0 rz 90 deg; joints [-2.371, -56.459, 89.196, 4.744, 18.345, -6.347]
  MoveL 715 to (-578.4, 300, 50) mm, rotated rx 180 ry 0 rz 90 deg; joints [-2.432, -58.492, 92.513, 5.22, 17.071, -6.882]
  MoveL 716 to (-578.4, 300, -0.5) mm, rotated rx 180 ry 0 rz 90 deg; joints [-2.432, -56.973, 93.038, 5.909, 15.036, -7.599]
  MoveL 717 to (-578.4, 300, 50) mm, rotated rx 180 ry 0 rz 90 deg; joints [-2.432, -58.492, 92.513, 5.22, 17.071, -6.882]
  MoveL 718 to (-578.4, 350, 50) mm, rotated rx 180 ry 0 rz 90 deg; joints [-2.497, -60.502, 95.739, 5.757, 15.865, -7.48]
  MoveL 719 to (-578.4, 350, -0.5) mm, rotated rx 180 ry 0 rz 90 deg; joints [-2.497, -58.929, 96.268, 6.612, 13.776, -8.365]
  MoveL 720 to (-578.4, 350, 50) mm, rotated rx 180 ry 0 rz 90 deg; joints [-2.497, -60.502, 95.739, 5.757, 15.865, -7.48]
  MoveL 721 to (-578.4, 400, 50) mm, rotated rx -180 ry 0 rz 90 deg; joints [-2.566, -62.495, 98.885, 6.364, 14.725, -8.151]
  MoveL 722 to (-578.4, 400, -0.5) mm, rotated rx -180 ry 0 rz 90 deg; joints [-2.566, -60.867, 99.419, 7.433, 12.579, -9.251]
  MoveL 723 to (-578.4, 400, 50) mm, rotated rx -180 ry 0 rz 90 deg; joints [-2.566, -62.495, 98.885, 6.364, 14.725, -8.151]
  MoveL 724 to (-578.4, 450, 50) mm, rotated rx -180 ry 0 rz 90 deg; joints [-2.638, -64.478, 101.958, 7.051, 13.65, -8.904]
  MoveL 725 to (-578.4, 450, -0.5) mm, rotated rx 180 ry 0 rz 90 deg; joints [-2.638, -62.791, 102.498, 8.396, 11.443, -10.282]
  MoveL 726 to (-578.4, 450, 50) mm, rotated rx -180 ry 0 rz 90 deg; joints [-2.638, -64.478, 101.958, 7.051, 13.65, -8.904]
  MoveL 727 to (-578.4, 500, 50) mm, rotated rx 180 ry 0 rz 90 deg; joints [-2.715, -66.457, 104.963, 7.829, 12.64, -9.752]
  MoveL 728 to (-578.4, 500, -0.5) mm, rotated rx 180 ry 0 rz 90 deg; joints [-2.715, -64.708, 105.511, 9.532, 10.369, -11.49]
  MoveL 729 to (-578.4, 500, 50) mm, rotated rx 180 ry 0 rz 90 deg; joints [-2.715, -66.457, 104.963, 7.829, 12.64, -9.752]
  MoveL 730 to (-578.4, 550, 50) mm, rotated rx 180 ry 0 rz 90 deg; joints [-2.796, -68.438, 107.907, 8.71, 11.696, -10.705]
  MoveL 731 to (-578.4, 550, -0.5) mm, rotated rx 180 ry 0 rz 90 deg; joints [-2.796, -66.624, 108.465, 10.882, 9.358, -12.914]
  MoveL 732 to (-578.4, 550, 50) mm, rotated rx 180 ry 0 rz 90 deg; joints [-2.796, -68.438, 107.907, 8.71, 11.696, -10.705]
  MoveL 733 to (-578.4, 600, 50) mm, rotated rx -180 ry 0 rz 90 deg; joints [-2.882, -70.427, 110.794, 9.704, 10.819, -11.775]
  MoveL 734 to (-578.4, 600, -0.5) mm, rotated rx 180 ry 0 rz 90 deg; joints [-2.882, -68.543, 111.363, 12.492, 8.412, -14.602]
  MoveL 735 to (-578.4, 600, 50) mm, rotated rx -180 ry 0 rz 90 deg; joints [-2.882, -70.427, 110.794, 9.704, 10.819, -11.775]
  MoveL 736 to (-578.4, 650, 50) mm, rotated rx 180 ry 0 rz 90 deg; joints [-2.973, -72.43, 113.629, 10.822, 10.013, -12.972]
  MoveL 737 to (-578.4, 650, -0.5) mm, rotated rx 180 ry 0 rz 90 deg; joints [-2.973, -70.472, 114.211, 14.418, 7.534, -16.61]
  MoveL 738 to (-578.4, 650, 50) mm, rotated rx 180 ry 0 rz 90 deg; joints [-2.973, -72.43, 113.629, 10.822, 10.013, -12.972]
  MoveL 739 to (-578.4, 700, 50) mm, rotated rx 180 ry 0 rz 90 deg; joints [-3.071, -74.453, 116.415, 12.067, 9.281, -14.301]
  MoveL 740 to (-578.4, 700, -0.5) mm, rotated rx -180 ry 0 rz 90 deg; joints [-3.071, -72.417, 117.011, 16.724, 6.728, -19.003]
  MoveL 741 to (-578.4, 700, 50) mm, rotated rx 180 ry 0 rz 90 deg; joints [-3.071, -74.453, 116.415, 12.067, 9.281, -14.301]
  MoveL 742 to (-578.4, 750, 50) mm, rotated rx 180 ry 0 rz 90 deg; joints [-3.175, -76.505, 119.154, 13.438, 8.627, -15.76]
  MoveL 743 to (-578.4, 750, -0.5) mm, rotated rx 180 ry 0 rz 90 deg; joints [-3.175, -74.385, 119.768, 19.475, 6.001, -21.845]
  MoveL 744 to (-578.4, 750, 50) mm, rotated rx 180 ry 0 rz 90 deg; joints [-3.175, -76.505, 119.154, 13.438, 8.627, -15.76]
  MoveL 745 to (-578.4, 800, 50) mm, rotated rx -180 ry 0 rz 90 deg; joints [-3.287, -78.593, 121.851, 14.919, 8.056, -17.333]
  MoveL 746 to (-578.4, 800, -0.5) mm, rotated rx 180 ry 0 rz 90 deg; joints [-3.287, -76.383, 122.483, 22.722, 5.36, -25.188]
  MoveL 747 to (-578.4, 800, 50) mm, rotated rx -180 ry 0 rz 90 deg; joints [-3.287, -78.593, 121.851, 14.919, 8.056, -17.333]
  MoveL 748 to (-578.4, 850, 50) mm, rotated rx -180 ry 0 rz 90 deg; joints [-3.406, -80.725, 124.506, 16.475, 7.576, -18.987]
  MoveL 749 to (-578.4, 850, -0.5) mm, rotated rx 180 ry 0 rz 90 deg; joints [-3.406, -78.419, 125.16, 26.473, 4.812, -29.041]
  MoveL 750 to (-578.4, 850, 50) mm, rotated rx -180 ry 0 rz 90 deg; joints [-3.406, -80.725, 124.506, 16.475, 7.576, -18.987]
  MoveL 751 to (-578.4, 900, 50) mm, rotated rx 180 ry 0 rz 90 deg; joints [-3.535, -82.912, 127.122, 18.049, 7.194, -20.664]
  MoveL 752 to (-578.4, 900, -0.5) mm, rotated rx -180 ry 0 rz 90 deg; joints [-3.535, -80.503, 127.8, 30.653, 4.365, -33.329]
  MoveL 753 to (-578.4, 900, 50) mm, rotated rx 180 ry 0 rz 90 deg; joints [-3.535, -82.912, 127.122, 18.049, 7.194, -20.664]
  MoveL 754 to (-578.4, 950, 50) mm, rotated rx 180 ry 0 rz 90 deg; joints [-3.674, -85.166, 129.7, 19.555, 6.919, -22.28]
  MoveL 755 to (-578.4, 950, -0.5) mm, rotated rx -180 ry 0 rz 90 deg; joints [-3.674, -82.645, 130.404, 35.046, 4.027, -37.836]
  MoveL 756 to (-578.4, 950, 50) mm, rotated rx 180 ry 0 rz 90 deg; joints [-3.674, -85.166, 129.7, 19.555, 6.919, -22.28]
  MoveL 757 to (-578.4, 1000, 50) mm, rotated rx 180 ry 0 rz 90 deg; joints [-3.824, -87.499, 132.241, 20.884, 6.761, -23.725]
  MoveL 758 to (-578.4, 1000, -0.5) mm, rotated rx -180 ry 0 rz 90 deg; joints [-3.824, -84.858, 132.976, 39.268, 3.802, -42.179]
  MoveL 759 to (-578.4, 1000, 50) mm, rotated rx 180 ry 0 rz 90 deg; joints [-3.824, -87.499, 132.241, 20.884, 6.761, -23.725]
  MoveL 760 to (-578.4, 1050, 50) mm, rotated rx -180 ry 0 rz 90 deg; joints [-3.986, -89.927, 134.745, 21.914, 6.732, -24.877]
  MoveL 761 to (-578.4, 1050, -0.5) mm, rotated rx -180 ry 0 rz 90 deg; joints [-3.986, -87.157, 135.514, 42.796, 3.692, -45.836]
  MoveL 762 to (-578.4, 1050, 50) mm, rotated rx -180 ry 0 rz 90 deg; joints [-3.986, -89.927, 134.745, 21.914, 6.732, -24.877]
  MoveL 763 to (-578.4, 1100, 50) mm, rotated rx 180 ry 0 rz 90 deg; joints [-4.164, -92.469, 137.213, 22.531, 6.848, -25.624]
  MoveL 764 to (-578.4, 1100, -0.5) mm, rotated rx -180 ry 0 rz 90 deg; joints [-4.164, -89.56, 138.02, 45.085, 3.699, -48.263]
  MoveL 765 to (-578.4, 1100, 50) mm, rotated rx 180 ry 0 rz 90 deg; joints [-4.164, -92.469, 137.213, 22.531, 6.848, -25.624]
  MoveL 766 to (-578.4, 1150, 50) mm, rotated rx -180 ry 0 rz 90 deg; joints [-4.357, -95.147, 139.644, 22.656, 7.13, -25.887]
  MoveL 767 to (-578.4, 1150, -0.5) mm, rotated rx -180 ry 0 rz 90 deg; joints [-4.357, -92.089, 140.494, 45.72, 3.829, -49.044]
  MoveL 768 to (-578.4, 1150, 50) mm, rotated rx -180 ry 0 rz 90 deg; joints [-4.357, -95.147, 139.644, 22.656, 7.13, -25.887]
